(* IEC 61131-3 sources: 1326_JeddahAppartment/1326 - Jeddah Appartment - Last/PLC1, 11 files *)

(* ---- PLC1.ST ---- *)
TYPE
  TCurtainStatus : Struct
    outUP   : BOOl;
    outDW   : BOOl;
    pos     : USINT;
    normPos : USINT;
  End_Struct;
END_TYPE

TYPE
   TEnCurtain : Struct
      UP   : BOOL;
      DW   : BOOl;
      STOP : BOOL;
   End_Struct;
END_TYPE

VAR_GLOBAL CONSTANT
   numOfCurtains      : USINT := 14;
   numOfCurtains_PLC1 : USINT := 9;
   numOfCurtains_PLC2 : USINT := 5;
END_VAR

VAR_GLOBAL
  curtainsStatus  AT PLC3.DATA : Array[1..numOfCurtains] of TCurtainStatus;
  PLC1_EnCurtains AT PLC1_Curtains.DATA : Array[1..numOfCurtains_PLC1] of TEnCurtain;
  PLC2_EnCurtains AT PLC2_Curtains.DATA : Array[1..numOfCurtains_PLC2] of TEnCurtain;
END_VAR

(* ---- fbControlFCU.ST ---- *)
Type
  TFCU_Mode      : (cooling, fanOnly);
  TFCU_FanSpeed  : (auto, low, med, high);

  TFCU_Settings  : Struct
     FCU_Mode     : TFCU_Mode;
     FCU_FanSpeed : TFCU_FanSpeed;
  End_Struct
End_Type

FUNCTION_BLOCK fbControlFCU
  VAR_INPUT
  enable   : BOOL;
  mode     : TFCU_Mode;      // 0  is cooling, 1 is fan only
  fanSpeed : TFCU_FanSpeed;  // 0 auto, 1 low, 2 med, 3 high
  setTemp  : REAL;
  temp     : REAL;
  END_VAR

  VAR_OUTPUT
  FCU_Status : TFCU_Status;
  END_VAR

  VAR_IN_OUT
  valve   : BOOL;
  fanLow  : BOOL;
  fanMed  : BOOl;
  fanHigh : BOOL;
  END_VAR

  VAR
  tempDiff : REAL;
  fanRotation_tick : fbTick;
  rotationTime : Time;
  END_VAR

  tempDiff := ABS(temp - setTemp);

  if not enable then
     valve := 0;
     FCU_Status.fanSpeed := 0;
  else
     if temp >= setTemp then
        if mode = cooling then
           valve := 1;
        else
           valve := 0;
        end_if;

        if fanSpeed <> auto then
           if fanSpeed = low then
              FCU_Status.fanSpeed := 1;
           elsif fanSpeed = med then
              FCU_Status.fanSpeed := 2;
           elsif fanSpeed = high then
              FCU_Status.fanSpeed := 4;
           end_if;
        else
           if tempDiff <= 2 then
              FCU_Status.fanSpeed := 1;
           elsif tempDiff >= 2.5 and tempDiff <= 4 then
              FCU_Status.fanSpeed := 2;
           elsif tempDiff >= 4.5 then
              FCU_Status.fanSpeed := 4;
           end_if;
        end_if;

     elsif temp < setTemp - 1 then
        valve := 0;
        if mode = fanOnly and fanSpeed <> auto then
           if fanSpeed = low then
              FCU_Status.fanSpeed := 1;
           elsif fanSpeed = med then
              FCU_Status.fanSpeed := 2;
           elsif fanSpeed = high then
              FCU_Status.fanSpeed := 4;
           end_if;
        else
           FCU_Status.fanSpeed := 0;
        end_if;
     end_if;
  end_if;

  fanLow  := FCU_Status.fanSpeed.0;
  fanMed  := FCU_Status.fanSpeed.1;
  fanHigh := FCU_Status.fanSpeed.2;

  FCU_Status.onOffStatus.0 := enable;
  FCU_Status.setTemp       := REAL_TO_INT(setTemp * 100);
  FCU_Status.roomTemp      := REAL_TO_INT(temp * 100);
  FCU_Status.valve.0       := valve;

  if mode = cooling then
     FCU_Status.mode := 0;
  elsif mode = fanOnly then
     FCU_Status.mode := 1;
  end_if;

  if fanSpeed = auto then
     FCU_Status.fanSpeedCtrl := 8;
  elsif fanSpeed = low then
     FCU_Status.fanSpeedCtrl := 1;
  elsif fanSpeed = med then
     FCU_Status.fanSpeedCtrl := 2;
  elsif fanSpeed = high then
     FCU_Status.fanSpeedCtrl := 4;
  end_if;

  if FCU_Status.fanSpeed = 0 then
     FCU_Status.fanRotationVar := 0;
  elsif FCU_Status.fanSpeed = 1 then
     rotationTime := T#0.5s;
  elsif FCU_Status.fanSpeed = 2 then
     rotationTime := T#0.25s;
  elsif FCU_Status.fanSpeed = 4 then
     rotationTime := T#0.1s;
  end_if;

  fanRotation_tick(IN := FCU_Status.fanSpeed <> 0, PT := rotationTime);

  if fanRotation_tick.Q then
     FCU_Status.fanRotationVar := UINT_TO_WORD(WORD_TO_UINT(FCU_Status.fanRotationVar) + 1);
  end_if;

  if FCU_Status.fanRotationVar = 6 then
     FCU_Status.fanRotationVar := 0;
  end_if;

END_FUNCTION_BLOCK

(* ---- fbControlHotelSystem_UDP.ST ---- *)
TYPE
  THotelPacket_Head : STRUCT
    frameHeader : WORD := 16#55AA;
    frameLength : UINT;
    SystemID    : DWORD := 16#41533354;
    cmdType     : Byte := 16#0F;
    frameNo     : WORD := 16#003A;
    nBuild      : BYTE := 16#FF;
    nUnit       : BYTE := 16#FF;
    nFloor      : BYTE := 16#FF;
    nRoom       : BYTE := 16#FF;
  END_STRUCT;
  TDevTypes :  (strongRelay := 1 , weakInput := 2 , weakOutput := 3 , serviceInfo := 4, curtainNode := 5,
              RS485Switch := 6, AirCond1 := 7, AirCond2 := 8, AirCond3 := 9, RS485Card := 10, RS485Heater := 11, EX_Relay := 14,
              IR := 15, EX_LED := 16, EX_Triac := 17, EX_RGB := 18, coreCtrl := 19, WeChatLock := 20, backMusic := 21,
              roomStateDimm := 22 , PMW_OUT := 23) ;

  TCtrlType : (open := 1, close := 2);

  TDevice : STRUCT
    DevType : TDevTypes;
    DevAddress : USINT ;
    loopAddress: UINT ;
    CtrlType   : TCtrlType := open;
    CtrlContent: USINT; (*from 0 to 100*)
  END_STRUCT;

  TDevCtrl : STRUCT
    NumOfDev : USINT := 1;
    DevArr : ARRAY [1..185] OF TDevice;
  END_STRUCT;

  THotelPacket : STRUCT
    Header : THotelPacket_Head;
    Data   : TDevCtrl;
    CRC    : UINT;
  END_STRUCT;

  TServerPacket : Struct
    userCode : Array[1..4] of byte := [0,0,0,0]; // keep zeros
    heartBeat: byte := 1;    // keep 1
    IP   :  TIPadr;
    port : UINT := 61000;
  END_Struct;

  TIamServerPacket : Struct
    Header         : THotelPacket_Head := (cmdType := 1 , frameNo := 16#000E);
    serverSettings : TServerPacket;
    CRC            : UINT;
  End_Struct;

  TAllStatusPacket : struct
    Header         : THotelPacket_Head;
    CRC            : UINT;
  End_struct;
END_TYPE

TYPE
   TDeviceStatus : STRUCT
    DevType : USINT;
    DevAddress : USINT ;
    loopAddress: UINT ;
    CtrlType   : BOOL;
    CtrlContent: USINT; (*from 0 to 100*)
  END_STRUCT;
END_TYPE

Type
    TBufferIn : Array[0..1349] of usint;
END_TYPE

FUNCTION_BLOCK fbControlHotelSystem_UDP
  VAR_INPUT

  RQ : BOOL;
  sendIamServer : BOOL R_EDGE;
  getAllStatus   : BOOL R_EDGE;
  ChanCode :  UINT;
  serverSettings : TServerPacket;

  END_VAR
  VAR_IN_OUT
  packet : THotelPacket;
  CH_IN : TBufferIn;
  END_vAR

  VAR_OUTPUT

  DevicesStatus : array[1..185] of TDeviceStatus;
  SysLock , cardType , Door : BOOl;
  numOfStatusDevs : uint;
  msgSent : BOOL;
  errCode : USINT;
  errText : STRING[100];
  END_VAR
  VAR
  IamServerPacket : TIamServerPacket;
  allStatusPacket : TAllStatusPacket;
  i : uint;
  index : uint;
  startIndex : UINT := 23;
  send_UDP : fbSendTO;
  CRC {Hidden} : PTR_TO UINT;
  END_VAR
  // OLD **** max controlled devices is 185 but the channel size must be max =  1350
  // In this project the channel length is modified in order to be able to create 7 channels
  // because when we crete 7 channels with 1350 bytes then the compiler reported allocation confilct error
  if not sendIamServer and not getAllStatus then
    if packet.Data.NumOfDev <= 0 then
       errCode := 65;
       errText := 'The number of devices is zero';
    elsif packet.Data.NumOfDev > 185 then
       errCode := 66;
       errText := 'The max number of devices is exceeded';
    else
      packet.Header.frameLength := SIZEOF(packet.Header) + 3 + (usint_to_uint(packet.Data.NumOfDev) * 6);
     // Length := packet.Header.frameLength;
      if packet.Header.frameLength <> 0 then
         if packet.Data.NumOfDev < 185  then
            CRC := adr(packet.Data.DevArr[packet.data.NumOfDev+1]);
            CRC^ := CheckCRC_16(ptr := adr(packet), length := packet.Header.frameLength - 2) ;
            packet.CRC := CRC^;
         elsif packet.Data.NumOfDev = 185 then
            packet.CRC := CheckCRC_16(ptr := adr(packet), length := packet.Header.frameLength - 2);
         end_if;
      end_if;
      send_UDP(rq := RQ, chanCode := ChanCode, lenTx := packet.Header.frameLength, data := void(packet) , mesSent => msgSent , error => errCode);
      errText := GetLastComErrTxt(errCode := errCode);
    end_if;
  elsif sendIamServer then
    IamServerPacket.Header.frameLength := SIZEOF(IamServerPacket) ;
    IamServerPacket.serverSettings := serverSettings;
    IamServerPacket.CRC := CheckCRC_16(ptr := adr(IamServerPacket), length := IamServerPacket.Header.frameLength - 2);

    send_UDP(rq := true, chanCode := ChanCode, lenTx := IamServerPacket.Header.frameLength, data := void(IamServerPacket) , mesSent => msgSent , error => errCode);
    errText := GetLastComErrTxt(errCode := errCode);
  elsif getAllStatus then
    allStatusPacket.Header.cmdType := 16#0E;
    allStatusPacket.Header.frameNo := 16#0001;
    allStatusPacket.Header.frameLength := SIZEOF(allStatusPacket);
    allStatusPacket.CRC := CheckCRC_16(ptr := adr(allStatusPacket), length := allStatusPacket.Header.frameLength - 2);

    send_UDP(rq := true, chanCode := ChanCode, lenTx := allStatusPacket.Header.frameLength, data := void(allStatusPacket) , mesSent => msgSent , error => errCode);
    errText := GetLastComErrTxt(errCode := errCode);
  end_if;

  // Read Status
  startIndex := 23;

  if CH_IN[8] = 14 then
    numOfStatusDevs := usint_to_uint(CH_IN[22]);
    for i := 1 to numOfStatusDevs  do
       index := startIndex + (i-1) * 6;
       DevicesStatus[i].DevType := CH_IN[index];
       DevicesStatus[i].DevAddress := CH_IN[index+1];
       DevicesStatus[i].loopAddress := USINT_TO_UINT(CH_IN[index+2]);
       if CH_IN[index+4] = 1 then
          DevicesStatus[i].CtrlType := true;
       elsif CH_IN[index+4] = 2 then
          DevicesStatus[i].CtrlType := false;
       end_if;
       DevicesStatus[i].CtrlContent := CH_IN[index+5];
    End_For;
    SysLock := usint_to_bool(CH_IN[15]);
    cardType := usint_to_bool(CH_IN[16]);
    Door  := usint_to_bool(CH_IN[17]);

  End_if;

END_FUNCTION_BLOCK

(* ---- fbControlRoom.ST ---- *)
Type
   TOutDev : struct
     DevAddress : USINT ;
     loopAddress: UINT ;
   End_Struct
End_Type

Type
  TLightsStatus         : Array[1..17] of BOOL ;
  TOutletsStatus        : Array[1..8]  of BOOL;
  TCurtainsUpStatus     : Array[1..6]  of BOOL;
  TCurtainsDwStatus     : Array[1..6]  of BOOL;
  TCurtainsFB           : Array[1..6]  of fb_iJalousie;
  TCurtainPositWm       : Array[1..6]  OF USINT;
  TMotionSensStatus     : Array[1..4]  of BOOL;
  TSwitchStatus         : Array[1..6]  of BOOL;

  TEnLights             : Array[1..17] of BOOL ;
  TEnLightsAN           : Array[1..17] of USINT; // 1:open  2:close 0:None
  //TEnLightsAN1          : USINT;
  TEnOutlets            : Array[1..8]  of BOOL;
  TEnOutletsAN          : Array[1..8]  of USINT; // 1:open  2:close 0:None
  TEnCurtainsUp         : Array[1..6]  of BOOL;
  TEnCurtainsDW         : Array[1..6]  of BOOL;

  TlightsOutputDevs     : Array[1..17] of TOutDev;
  ToutletOutputDevs     : Array[1..8]  of TOutDev;
  TcurtainsUpOutputDevs : Array[1..6]  of TOutDev;
  TcurtainsDwOutputDevs : Array[1..6]  of TOutDev;
  TMotionSensOutputDevs : Array[1..4]  of TOutDev;
  TExRelayAdd           : ARRAY[1..2]  OF USINT;

End_Type

FUNCTION_BLOCK fbControlRoom
(*function block that send the command to RCU to control
the lights, curtains, and outlets
*)
  VAR_INPUT
    RCU_ChCode       : UINT;
   // RCU_ethAdrToSet  : TRemoteEthAdr;

   // RCU_IP_toSet     : TIPadr;

    numOfLights      : USINT;
    numOfOutlets     : USINT;
    numOfCurtains    : USINT;
    numOfMotionSens  : USINT;
    RCU_PingDone     : BOOL;

    lightsOutputDevs      : TlightsOutputDevs;
    outletOutputDevs      : ToutletOutputDevs;
    curtainsUpOutputDevs  : TcurtainsUpOutputDevs;
    curtainsDwOutputDevs  : TcurtainsDwOutputDevs;
    MotionSensOutputDevs  : TMotionSensOutputDevs;

  END_VAR
  VAR_OUTPUT
  //    CurtainPositWm   : TCurtainPositWm;

      ExRelay1_LVO : array[1..24] of TDeviceStatus;
      ExRelay2_LVO : array[1..24] of TDeviceStatus;

      SwitchUPStatus  : TSwitchStatus;
      SwitchDWStatus  : TSwitchStatus;
  END_VAR
  VAR_IN_OUT
    RCU_CH_IN     : TBufferIn;
 //   Set_IP           : BOOL;

    LightsStatus     : TLightsStatus;
    OutletsStatus    : TOutletsStatus;
  //  CurtainsUpStatus : TCurtainsUpStatus;
  //  CurtainsDwStatus : TCurtainsDwStatus;
  //  CurtainsFB       : TCurtainsFB;
    MotionSenStatus  : TMotionSensStatus;

    EnLights       : TEnLights     ;
    EnLightsAN     : TEnLightsAN   ;
   // EnLightsAN1  : TEnLightsAN1;
    EnOutlets      : TEnOutlets    ;
    EnOutletsAN    : TEnOutletsAN   ;
  //  EnCurtainsUp   : TEnCurtainsUp ;
  //  EnCurtainsDw   : TEnCurtainsDW ;

    SendIamServer : BOOL;
    GetAllStatus  : BOOL;

  END_VAR
  VAR
    RCU           : fbControlHotelSystem_UDP;
    RCU_RQ        : BOOL;
    Server_settings  : TServerPacket := (IP := [192,168,0,16])  ;
    sentPacket       : THotelPacket;
    K : USINT;
    i : UINT;
    cmd_CtrlType     : TCtrlType  ;
    cmd_CtrlContent  : USINT;
    cmd_CtrlType1    : TCtrlType  ;
    cmd_CtrlContent1 : USINT;

    TonCurtainsWait : Array[1..5]  of TON ;
    EnCurtainsWait  : Array[1..5]  of BOOL ;
    //TpCurtains      : Array[1..5]  of TPR;
    EnCurtains      : Array[1..5]  of BOOL ;
    //ReCurtainsTp    : Array[1..5]  of BOOL ;
    RTCurtains      : Array[1..5]  of R_TRIG;
    FTCurtains      : Array[1..5]  of F_TRIG;
    Up              : Array[1..5]  of BOOL ;
    Dw              : Array[1..5]  of BOOL ;
    NumOfCmd        : USINT := 1;
    RCU_Connected   : BOOL;

    RCU_Connected_RT : R_TRIG;
    RCU_Connection_TOF : TOF;
    restorStatusDone      : BOOL;
    test                  : USINT;
    PlcEthAdr             : TlocalEthAdr ;
    RCU_ChAdr             : TRemoteEthAdr;

  END_VAR

//  IF Set_IP THEN
//     SetRemoteIPaddress(rq := True , chanCode :=RCU_ChCode , ethAdr :=RCU_ethAdrToSet ) ;
//     Set_IP := 0 ;
//  END_IF;

   for i := 1 to RCU.numOfStatusDevs do

      if RCU.DevicesStatus[i].DevType = 6 and RCU.DevicesStatus[i].DevAddress = 1 then
        ExRelay1_LVO[RCU.DevicesStatus[i].loopAddress] := RCU.DevicesStatus[i];

      elsif RCU.DevicesStatus[i].DevType = 6 and RCU.DevicesStatus[i].DevAddress = 2 then
        ExRelay2_LVO[RCU.DevicesStatus[i].loopAddress] := RCU.DevicesStatus[i];
      end_if;

   End_for;

  if GetIPaddress(ethChan := ETH1 , ethAdr := PlcEthAdr) then
     Server_settings.IP := PlcEthAdr.IP ;
  end_if;

  if GetRemoteIPaddress(chanCode := RCU_ChCode, ethAdr := RCU_ChAdr) then
     Server_settings.port := RCU_ChAdr.localPort ;
  end_if;

  RCU(RQ := RCU_RQ , sendIamServer :=SendIamServer , getAllStatus := GetAllStatus , ChanCode := RCU_ChCode , serverSettings := Server_settings , packet := sentPacket, CH_IN := RCU_CH_IN);

  IF RCU.msgSent THEN
    RCU_RQ := 0 ;
    SendIamServer := 0 ;
    GetAllStatus  := 0 ;
    NumOfCmd := 1 ;
    restorStatusDone :=0;
  END_IF;

  RCU_Connection_TOF(IN := RCU_PingDone , PT :=T#1s , Q => RCU_Connected );
  RCU_Connected_RT(CLK := RCU_Connected );

  IF RCU_Connected_RT.Q THEN
    restorStatusDone :=1;
  END_IF;
  IF IS_COLD_RESTART_PLC OR IS_HOT_RESTART_PLC THEN
     GetAllStatus :=1;
  END_IF;
  IF restorStatusDone THEN
     if numOfLights > 0 then
       FOR K := 1 TO numOfLights DO
          IF LightsStatus[K] THEN
            cmd_CtrlType := open ;
            cmd_CtrlContent := 100 ;
          ELSE
            cmd_CtrlType := close ;
            cmd_CtrlContent := 0 ;
          END_IF;
          sentPacket.Data.DevArr[NumOfCmd].DevType     := EX_Relay ;
          sentPacket.Data.DevArr[NumOfCmd].DevAddress  := lightsOutputDevs[K].DevAddress;
          sentPacket.Data.DevArr[NumOfCmd].loopAddress := lightsOutputDevs[K].loopAddress ;
          sentPacket.Data.DevArr[NumOfCmd].CtrlType    := cmd_CtrlType ;
          sentPacket.Data.DevArr[NumOfCmd].CtrlContent := cmd_CtrlContent ;
          NumOfCmd := NumOfCmd + 1 ;
          test := test + 1 ;
       END_FOR;
     end_if;

     if numOfOutlets > 0 then
       FOR K := 1 TO numOfOutlets DO
          IF OutletsStatus[K] THEN
            cmd_CtrlType := open ;
            cmd_CtrlContent := 100 ;
          ELSE
            cmd_CtrlType := close ;
            cmd_CtrlContent := 0 ;
          END_IF;
          sentPacket.Data.DevArr[NumOfCmd].DevType     := EX_Relay ;
          sentPacket.Data.DevArr[NumOfCmd].DevAddress  := outletOutputDevs[K].DevAddress;
          sentPacket.Data.DevArr[NumOfCmd].loopAddress := outletOutputDevs[K].loopAddress ;
          sentPacket.Data.DevArr[NumOfCmd].CtrlType    := cmd_CtrlType ;
          sentPacket.Data.DevArr[NumOfCmd].CtrlContent := cmd_CtrlContent ;
          NumOfCmd := NumOfCmd + 1 ;
       END_FOR;
     end_if;
     sentPacket.Data.NumOfDev := NumOfCmd ;
     RCU_RQ := 1 ;
     restorStatusDone := 0;
    // GetAllStatus := 1;
  ELSE
    FOR i := 1 to RCU.numOfStatusDevs DO
       IF RCU.DevicesStatus[i].DevType = 14 THEN
         if numOfLights > 0 then
           FOR K := 1 TO numOfLights DO
             IF RCU.DevicesStatus[i].loopAddress = lightsOutputDevs[K].loopAddress AND RCU.DevicesStatus[i].DevAddress = lightsOutputDevs[K].DevAddress THEN
                lightsStatus[K] := RCU.DevicesStatus[i].CtrlType;
             END_IF;
           END_FOR;
         end_if;

         if numOfOutlets > 0 then
           FOR K := 1 TO numOfOutlets DO
             IF RCU.DevicesStatus[i].loopAddress = outletOutputDevs[K].loopAddress AND RCU.DevicesStatus[i].DevAddress = outletOutputDevs[k].DevAddress THEN
                outletsStatus[K] := RCU.DevicesStatus[i].CtrlType;
             END_IF;
           END_FOR;
         end_if;
        (* FOR K := 1 TO numOfCurtains DO
           IF RCU.DevicesStatus[i].loopAddress = curtainsUpOutputDevs[K].loopAddress AND RCU.DevicesStatus[i].DevAddress = curtainsUpOutputDevs[K].DevAddress  THEN
              CurtainsUpStatus[K] := RCU.DevicesStatus[i].CtrlType;
           END_IF;
         END_FOR;
         FOR K := 1 TO numOfCurtains DO
           IF RCU.DevicesStatus[i].loopAddress = curtainsDwOutputDevs[K].loopAddress AND RCU.DevicesStatus[i].DevAddress = curtainsDwOutputDevs[K].DevAddress THEN
              CurtainsDwStatus[K] := RCU.DevicesStatus[i].CtrlType;
           END_IF;
         END_FOR; *)

       ELSIF RCU.DevicesStatus[i].DevType = 6 THEN

         // get the status of motion sensors
         if numOfMotionSens > 0 then
           FOR K := 1 TO numOfMotionSens  DO
             IF RCU.DevicesStatus[i].loopAddress = MotionSensOutputDevs[K].loopAddress AND RCU.DevicesStatus[i].DevAddress = MotionSensOutputDevs[K].DevAddress THEN
                MotionSenStatus[K] := RCU.DevicesStatus[i].CtrlType;
             END_IF;
           END_FOR;
         end_if;

         // Get the status of switch keys from the RCU
         if numOfCurtains > 0 then
           FOR K := 1 TO numOfCurtains  DO
             IF RCU.DevicesStatus[i].loopAddress = curtainsUpOutputDevs[K].loopAddress AND RCU.DevicesStatus[i].DevAddress = curtainsUpOutputDevs[K].DevAddress THEN
                SwitchUPStatus[K] := RCU.DevicesStatus[i].CtrlType;
             END_IF;

             IF RCU.DevicesStatus[i].loopAddress = curtainsDwOutputDevs[K].loopAddress AND RCU.DevicesStatus[i].DevAddress = curtainsDwOutputDevs[K].DevAddress THEN
                SwitchDWStatus[K] := RCU.DevicesStatus[i].CtrlType;
             END_IF;
           END_FOR;
         end_if;

       END_IF;
    END_FOR;
  END_IF;

  //FOR test
  (*IF (EnLightsAN1 = 1 AND LightsStatus[1] = false) OR (EnLightsAN1 = 2 AND LightsStatus[1] = true) THEN
      EnLights[1]   := 1;
      EnLightsAN1 := 0;
  ELSE
      EnLightsAN1 :=0;
  END_IF;*)

  if numOfLights > 0 then
    FOR K := 1 TO numOfLights DO
       IF (EnLightsAN[K] = 1 AND LightsStatus[K] = false) OR (EnLightsAN[K] = 2 AND LightsStatus[K] = true) THEN
          EnLights[K]   := 1;
          EnLightsAN[K] := 0;
       ELSE
          EnLightsAN[K] :=0;
       END_IF;

       IF EnLights[K] THEN
         EnLights[K] := 0 ;
         IF lightsStatus[K] THEN
            cmd_CtrlType     := close ;
            cmd_CtrlContent  := 0 ;
         ELSE
            cmd_CtrlType     := open ;
            cmd_CtrlContent  := 100 ;
         END_IF;
         sentPacket.Data.NumOfDev := 1 ;
         sentPacket.Data.DevArr[1].DevType := EX_Relay ;
         sentPacket.Data.DevArr[1].DevAddress := lightsOutputDevs[K].DevAddress;
         sentPacket.Data.DevArr[1].loopAddress := lightsOutputDevs[K].loopAddress ;
         sentPacket.Data.DevArr[1].CtrlType := cmd_CtrlType ;
         sentPacket.Data.DevArr[1].CtrlContent := cmd_CtrlContent ;
         RCU_RQ :=1;
       END_IF;
    END_FOR;
  end_if;

  if numOfOutlets > 0 then
    FOR K := 1 TO numOfOutlets DO
       IF (EnOutletsAN[K] = 1 AND OutletsStatus[K] = false) OR (EnOutletsAN[K] = 2 AND OutletsStatus[K] = true) THEN
          EnOutlets[K]   := 1;
          EnOutletsAN[K] := 0;
       ELSE
          EnOutletsAN[K] := 0;
       END_IF;

       IF EnOutlets[K] THEN
         EnOutlets[K] := 0 ;
         IF outletsStatus[K] THEN
            cmd_CtrlType     := close ;
            cmd_CtrlContent  := 0 ;
         ELSE
            cmd_CtrlType     := open ;
            cmd_CtrlContent  := 100 ;
         END_IF;
         sentPacket.Data.NumOfDev := 1 ;
         sentPacket.Data.DevArr[1].DevType := EX_Relay ;
         sentPacket.Data.DevArr[1].DevAddress := outletOutputDevs[K].DevAddress;
         sentPacket.Data.DevArr[1].loopAddress := outletOutputDevs[K].loopAddress ;
         sentPacket.Data.DevArr[1].CtrlType := cmd_CtrlType ;
         sentPacket.Data.DevArr[1].CtrlContent := cmd_CtrlContent ;
         RCU_RQ :=1;
       END_IF;
    END_FOR;
  end_if;

   (*
   FOR K := 1 TO numOfCurtains DO
      IF ((EnCurtainsUp[K] AND Dw[K]) OR (EnCurtainsDw[K] AND Up[K])) THEN
       EnCurtains[K] := 0;
       curtainsFB[k](stop := 1  , upDwTime :=T#20s );

       sentPacket.Data.NumOfDev := 2 ;
       sentPacket.Data.DevArr[1].DevType := EX_Relay ;
       sentPacket.Data.DevArr[1].DevAddress := curtainsUpOutputDevs[K].DevAddress;
       sentPacket.Data.DevArr[1].loopAddress := curtainsUpOutputDevs[K].loopAddress ;
       sentPacket.Data.DevArr[1].CtrlType := close ;
       sentPacket.Data.DevArr[1].CtrlContent := 0 ;

       sentPacket.Data.DevArr[2].DevType := EX_Relay ;
       sentPacket.Data.DevArr[2].DevAddress := curtainsDwOutputDevs[K].DevAddress;
       sentPacket.Data.DevArr[2].loopAddress := curtainsDwOutputDevs[K].loopAddress ;
       sentPacket.Data.DevArr[2].CtrlType := close ;
       sentPacket.Data.DevArr[2].CtrlContent := 0 ;
       RCU_RQ :=1;

       Up[K] := EnCurtainsUp[K] ;
       Dw[K] := EnCurtainsDw[K] ;
       EnCurtainsUp[K] := 0;
       EnCurtainsDw[K] := 0;
       EnCurtainsWait[K] := 1;
    ELSIF (EnCurtainsUp[K] AND Dw[K] = false ) OR (EnCurtainsDw[K] AND Up[K] = false ) THEN
     //  IF curtainsFB[K].posit > 0 THEN
          Up[K] := EnCurtainsUp[K] ;
          EnCurtains[K]   := 1;
     //  ELSIF curtainsFB[K].posit < 100 THEN
          Dw[K] := EnCurtainsDw[K] ;
       //   EnCurtains[K]   := 1;
    //   END_IF;
       EnCurtainsUp[K] := 0;
       EnCurtainsDw[K] := 0;

    END_IF;

    TonCurtainsWait[K](IN := EnCurtainsWait[K] , PT := T#1s );
     IF TonCurtainsWait[K].Q THEN
       EnCurtainsWait[K] := 0;
       EnCurtains[K] := 1;
     END_IF;

     IF EnCurtains[K] THEN
        curtainsFB[K](up := CurtainsUpStatus[K] , dw := CurtainsDwStatus[K]  , upDwTime :=T#20s );
     END_IF;

     IF (curtainsFB[K].posit = 0 and curtainsFB[K].outUp) OR (curtainsFB[K].posit = 100 and curtainsFB[K].outDw) THEN
        EnCurtains[K] := 0;
        Up[K] := 0;
        Dw[K] := 0;
        curtainsFB[K](stop := 1  , upDwTime :=T#20s );
     END_IF;

     IF CurtainsFB[K].posit = 0 THEN
        CurtainPositWm[k] := 0;
     ELSIF CurtainsFB[K].posit > 0 AND CurtainsFB[K].posit < 30 THEN
        CurtainPositWm[K] := 1;
     ELSIF CurtainsFB[K].posit >= 30 AND CurtainsFB[K].posit < 60 THEN
        CurtainPositWm[K] := 2;
     ELSIF CurtainsFB[K].posit >= 60 AND CurtainsFB[K].posit < 90  THEN
        CurtainPositWm[K] := 3;
     ELSIF CurtainsFB[K].posit >= 100 THEN
        CurtainPositWm[K] := 4;
     END_IF;
     IF Up[K] THEN
        cmd_CtrlType    := open;
        cmd_CtrlContent := 100;
     ELSE
        cmd_CtrlType    := close;
        cmd_CtrlContent := 0;
     END_IF;
     IF Dw[K] THEN
        cmd_CtrlType1    := open;
        cmd_CtrlContent1 := 100;
     ELSE
        cmd_CtrlType1    := close;
        cmd_CtrlContent1 := 0;
     END_IF;
     RTCurtains[K](CLK := EnCurtains[K] ) ;
     FTCurtains[K](CLK := EnCurtains[K] ) ;
     IF RTCurtains[K].Q OR FTCurtains[K].Q THEN
       sentPacket.Data.NumOfDev := 2 ;
       sentPacket.Data.DevArr[1].DevType     := EX_Relay ;
       sentPacket.Data.DevArr[1].DevAddress  := curtainsUpOutputDevs[K].DevAddress;
       sentPacket.Data.DevArr[1].loopAddress := curtainsUpOutputDevs[K].loopAddress ;
       sentPacket.Data.DevArr[1].CtrlType    := cmd_CtrlType ;
       sentPacket.Data.DevArr[1].CtrlContent := cmd_CtrlContent ;

       sentPacket.Data.DevArr[2].DevType     := EX_Relay ;
       sentPacket.Data.DevArr[2].DevAddress  := curtainsDwOutputDevs[K].DevAddress;
       sentPacket.Data.DevArr[2].loopAddress := curtainsDwOutputDevs[K].loopAddress ;
       sentPacket.Data.DevArr[2].CtrlType    := cmd_CtrlType1 ;
       sentPacket.Data.DevArr[2].CtrlContent := cmd_CtrlContent1 ;
       RCU_RQ :=1;
     END_IF;
   END_FOR;  *)

END_FUNCTION_BLOCK

(* ---- PrgConnectHMIs.ST ---- *)
Type
  T_HMI_Info : struct
     SNo          : USINT;
     readStAdd    : UINT;
     writeStAdd   : UINT;
     readNoPoint  : UINT;
     writeNoPoint : UINT;
  End_Struct;

  //================= Read from HMI =================

  TShutterControl : struct
     Dw : WORD;
     UP : WORD;
  End_Struct;

  TFCU_Control : struct
     onOff       : WORD;
     SetTempCtrl : WORD; //  bit 0 for increment, bit 1 for decrement
     setTemp     : INT;
     fanSpeed    : WORD;
     mode        : WORD;
  End_Struct;

  T_HMI_DataRead : struct
     enLights   : Array[1..17] of WORD;
     enOutlets  : Array[1..8] of WORD;
     enShutters : Array[1..6] of TShutterControl;
     enFCUs     : Array[1..3] of TFCU_Control;
  End_Struct;

  //================= Write To HMI ==================

  TShutterStatus : struct
     Dw  : WORD;
     UP  : WORD;
     pos : WORD;
  End_Struct;

  TFCU_Status  : Struct
     onOffStatus    : WORD;
     setTemp        : INT;
     roomTemp       : INT;
     fanSpeed       : WORD;
     mode           : WORD;
     valve          : WORD;
     fanSpeedCtrl   : WORD;
     fanRotationVar : WORD;   // var for rotating the fan GIF in the HMI according to the current fan speed
  End_Struct;

  T_HMI_DataWrite : struct
     lightsStatus     : Array[1..17] of WORD;
     outletsStatus    : Array[1..8]  of WORD;
     motionSensStatus : Array[1..4]  of WORD;
     shuttersStatus   : Array[1..6]  of TShutterStatus;
     FCUs_Status      : Array[1..3]  of TFCU_Status;
  End_Struct;

End_Type

Var_Global Constant
   numOfHMIs : INT := 10;
   //HMIs_Info : Array[1..numOfHMIs] of T_HMI_Info := [()];
End_Var

Var_Global Retain
   HMIs_DataRead  : Array[1..numOfHMIs] of T_HMI_DataRead;     // Data is read from HMI
   HMIs_DataWrite : Array[1..numOfHMIs] of T_HMI_DataWrite;    // Data is written to HMI

   HMIs_Info : Array[1..numOfHMIs] of T_HMI_Info := [()];
End_Var

Var_Global
  cmdArr : Array[1..numOfHMIs * 2] of TCmdStruct;
  GrSel  : USINT ;
End_Var

PROGRAM PrgConnectHMIs
  VAR_INPUT
  END_VAR
  VAR_OUTPUT
  END_VAR
  VAR
  master : fbModbusRTUmas2;
  //cmdArr : Array[1..numOfHMIs * 2] of TCmdStruct;

  i      : INT ;
  maxCmd : USINT;

  END_VAR
  VAR_TEMP
  END_VAR

  if IS_COLD_RESTART_PLC or IS_HOT_RESTART_PLC then
     GrSel := 2;
  end_if;

  for i := 1 to numOfHMIs do
      ModbusCmd(Gr := 2, SNo := HMIs_Info[i].SNo, FNC := 3,  StAdr := HMIs_Info[i].readStAdd,   NoPoint := HMIs_Info[i].readNoPoint, PtrData := adr(HMIs_DataRead[i]), Cmd := cmdArr[i*2-1]) ;

      ModbusCmd(Gr := 2, SNo := HMIs_Info[i].SNo, FNC := 16, StAdr := HMIs_Info[i].writeStAdd , NoPoint := HMIs_Info[i].writeNoPoint, PtrData := adr(HMIs_DataWrite[i]), Cmd := cmdArr[i*2]) ;
  end_for;

  //maxCmd := INT_TO_USINT(numOfHMIs * 2);

  maxCmd := 2;
  master(EN := true, GrSel := GrSel,  MaxCmd := maxCmd , chanCode := CH2_uni , Delay := T#0.2s, Commands := cmdArr[9], MBtimeOut := T#0.5s);

END_PROGRAM

(* ---- PrgInterance.ST ---- *)
VAR_GLOBAL CONSTANT
   NumOfLightInterance      : USINT := 6;
   NumOfOutletInterance     : USINT := 2;
   NumOfCurtainInterance    : USINT := 0;
   NumOfMotionSensInterance : USINT := 1;
   NumOfFCUsInterance       : USINT := 0;
   NumOfHMIsInterance       : USINT := 1;
END_VAR

VAR_GLOBAL RETAIN
   lightsStatusInterance  {PUBLIC_API} : TLightsStatus;
   outletsStatusInterance {PUBLIC_API} : TOutletsStatus;
 (*  setTempFCU_Interance  : Array[1..NumOfFCUsInterance] of REAL := [20];
  *)

END_VAR

PROGRAM PrgInterance

  VAR
  //WebMaker
  lightsSelect   : BOOL;
  socketsSelect  : BOOL;
  shuttersSelect : BOOL;
  AC_Select      : BOOL;
  navSelect      : usint;

  //RCU
  RCU_ethAdr   : TRemoteEthAdr;
  RCU_IP : TIPadr := [192, 168, 0, 23];
  RCU_Ch_localPort : UINT;
  Set_IP           : BOOL;
  GetAllStatus  : BOOL;
  SendIamServer : BOOL;

  //controlRoom
  controlRoom   : fbControlRoom ;
  lightsOutputDevs     : TlightsOutputDevs     := [(DevAddress := 1 , loopAddress := 1),(DevAddress := 1 , loopAddress := 2),
                                                   (DevAddress := 1 , loopAddress := 3),(DevAddress := 1 , loopAddress := 4),
                                                   (DevAddress := 1 , loopAddress := 5),(DevAddress := 1 , loopAddress := 6)];

  outletOutputDevs     : ToutletOutputDevs     := [(DevAddress := 1 , loopAddress := 7)];

  (*curtainsUpOutputDevs : TcurtainsUpOutputDevs := [(DevAddress := 1 , loopAddress := 8)];
  curtainsDwOutputDevs : TcurtainsDwOutputDevs := [(DevAddress := 1 , loopAddress := 9)];*)

  motionSensOutputDevs : TMotionSensOutputDevs := [(DevAddress := 1 , loopAddress := 1)];

  EnLights                            : TEnLights     ;
  EnLightsAN       {PUBLIC_API}       : TEnLightsAN   ;
  EnOutlets                           : TEnOutlets    ;
  EnOutletsAN      {PUBLIC_API}       : TEnOutletsAN  ;
  EnCurtainsUp     {PUBLIC_API}       : TEnCurtainsUp ;
  EnCurtainsDw     {PUBLIC_API}       : TEnCurtainsDW ;
   //EnLightsInteranceAN1  {PUBLIC_API}      : TEnLightsAN1    ;
   //stLightsInteranceAN  {PUBLIC_API}       : BOOL     ;
  //curtainsFB       : TCurtainsFB;
  //CurtainPositWm   : TCurtainPositWm;

  //
  enLights_RT  : Array[1..NumOfHMIsInterance,1..NumOfLightInterance] of R_TRIG;
  enLights_FT  : Array[1..NumOfHMIsInterance,1..NumOfLightInterance] of F_TRIG;

  enOutlets_RT : Array[1..NumOfHMIsInterance,1..NumOfOutletInterance] of R_TRIG;
  enOutlets_FT : Array[1..NumOfHMIsInterance,1..NumOfOutletInterance] of F_TRIG;
  (*
  enCurtainsUP_RT : Array[1..NumOfHMIsInterance,1..NumOfCurtainInterance] of R_TRIG;
  enCurtainsUP_FT : Array[1..NumOfHMIsInterance,1..NumOfCurtainInterance] of F_TRIG;

  enCurtainsDW_RT : Array[1..NumOfHMIsInterance,1..NumOfCurtainInterance] of R_TRIG;
  enCurtainsDW_FT : Array[1..NumOfHMIsInterance,1..NumOfCurtainInterance] of F_TRIG; *)

  //
  i , j : USINT;
  afterRestart_TP : TP;
  afterRestart_TP_FT : F_TRIG;

  //
  motionSensStatus                : TMotionSensStatus;
  CurtainsUpStatus   {PUBLIC_API} : TCurtainsUpStatus;
  CurtainsDwStatus   {PUBLIC_API} : TCurtainsDwStatus;

  // FCU VARS
  (*FCU          : Array[1..NumOfFCUsInterance] of fbControlFCU;
  enableFCU    : Array[1..NumOfFCUsInterance] of BOOL;
  settingsFCU  : Array[1..NumOfFCUsInterance] of TFCU_Settings;

  //modeFCU      : Array[1..NumOfFCUsInterance] of TFCU_Mode;
  //fanSpeedFCU  : Array[1..NumOfFCUsInterance] of TFCU_FanSpeed;

  enFCUs_FT    : Array[1..NumOfHMIsInterance,1..NumOfFCUsInterance] of F_TRIG;
  enFCUs_RT    : Array[1..NumOfHMIsInterance,1..NumOfFCUsInterance] of R_TRIG;

  enFanHigh_RT : Array[1..NumOfHMIsInterance,1..NumOfFCUsInterance] of R_TRIG;
  enFanMed_RT  : Array[1..NumOfHMIsInterance,1..NumOfFCUsInterance] of R_TRIG;
  enFanLow_RT  : Array[1..NumOfHMIsInterance,1..NumOfFCUsInterance] of R_TRIG;
  enFanAuto_RT : Array[1..NumOfHMIsInterance,1..NumOfFCUsInterance] of R_TRIG;

  enFCUCool_RT    : Array[1..NumOfHMIsInterance,1..NumOfFCUsInterance] of R_TRIG;
  enFCUFanOnly_RT : Array[1..NumOfHMIsInterance,1..NumOfFCUsInterance] of R_TRIG;

  enSetTempIncr_RT : Array[1..NumOfHMIsInterance,1..NumOfFCUsInterance] of R_TRIG;
  enSetTempIncr_FT : Array[1..NumOfHMIsInterance,1..NumOfFCUsInterance] of F_TRIG;

  enSetTempDecr_RT : Array[1..NumOfHMIsInterance,1..NumOfFCUsInterance] of R_TRIG;
  enSetTempDecr_FT : Array[1..NumOfHMIsInterance,1..NumOfFCUsInterance] of F_TRIG;  *)

  //HMIs[1..num
  HMI_Index : USINT;
  RCU_Index : USINT;
  HMI_Addresses : Array[1..NumOfHMIsInterance] of USINT := [1];

  END_VAR

  if navSelect = 0 then
     lightsSelect   := 1;
     socketsSelect  := 0;

  elsif navSelect = 1 then
     lightsSelect   := 0;
     socketsSelect  := 1;
  end_if;

  HMI_Index := 1;
  RCU_Index := 1;

  if GetRemoteIPaddress(chanCode := Eth1_uni0, ethAdr := RCU_ethAdr) then
     RCUs_IPs[RCU_Index] := RCU_ethAdr.remoteIP;
  end_if;

  HMIs_Info[HMI_Index].SNo := HMI_Addresses[1];
  HMIs_Info[HMI_Index].readStAdd  := 131;
  HMIs_Info[HMI_Index].writeStAdd := 191;
  HMIs_Info[HMI_Index].readNoPoint  := SIZEOF(HMIs_DataRead[HMI_Index]) / 2;
  HMIs_Info[HMI_Index].writeNoPoint := SIZEOF(HMIs_DataWrite[HMI_Index]) / 2;

  for i := 1 to NumOfHMIsInterance-1 do
    HMIs_Info[HMI_Index+i] := HMIs_Info[HMI_Index];
    HMIs_Info[HMI_Index+i].SNo := HMI_Addresses[i+1];
  end_for;

  afterRestart_TP(IN := IS_COLD_RESTART_PLC or IS_HOT_RESTART_PLC, PT := T#2s );
  afterRestart_TP_FT(CLK := afterRestart_TP.Q);

  if afterRestart_TP_FT.Q then
     SendIamServer := 1;
  end_if;

  controlRoom(RCU_ChCode := ETH1_uni0 , RCU_PingDone := RCUs_PingDone[RCU_Index],
              numOfLights := NumOfLightInterance , numOfOutlets := NumOfOutletInterance , numOfCurtains := 0, numOfMotionSens := NumOfMotionSensInterance,
              lightsOutputDevs := lightsOutputDevs , outletOutputDevs := outletOutputDevs ,
              RCU_CH_IN := void(ETH1_uni0_IN) , LightsStatus := lightsStatusInterance ,OutletsStatus := outletsStatusInterance, MotionSenStatus := motionSensStatus,
              EnLights := EnLights , EnLightsAN := EnLightsAN , EnOutlets := EnOutlets ,EnOutletsAN :=EnOutletsAN ,
              SendIamServer := SendIamServer , GetAllStatus := GetAllStatus);

              //stLightsInteranceAN := lightsStatusInterance[1];

   for i := 1 to NumOfLightInterance do
       HMIs_DataWrite[HMI_Index].lightsStatus[i] := BOOL_TO_WORD(lightsStatusInterance[i]);
   end_for;

   for i := 1 to NumOfOutletInterance do
       HMIs_DataWrite[HMI_Index].outletsStatus[i] := BOOL_TO_WORD(outletsStatusInterance[i]);
   end_for;

   for i := 1 to NumOfMotionSensInterance do
       HMIs_DataWrite[HMI_Index].motionSensStatus[i] := BOOL_TO_WORD(motionSensStatus[i]);
   end_for;

   for j := 1 to NumOfHMIsInterance do
     for i := 1 to NumOfLightInterance do

         enLights_RT[j,i](CLK := HMIs_DataRead[HMI_Index + j - 1].enLights[i]);

         enLights_FT[j,i](CLK := HMIs_DataRead[HMI_Index + j - 1].enLights[i]);

         if enLights_RT[j,i].Q or enLights_FT[j,i].Q then
            EnLights[i] := 1;
         end_if;
     end_for;
   end_for;

   for j := 1 to NumOfHMIsInterance do
     for i := 1 to NumOfOutletInterance do

         enOutlets_RT[j,i](CLK := HMIs_DataRead[HMI_Index + j - 1].enOutlets[i]);

         enOutlets_FT[j,i](CLK := HMIs_DataRead[HMI_Index + j - 1].enOutlets[i]);

         if enOutlets_RT[j,i].Q or enOutlets_FT[j,i].Q then
            EnOutlets[i] := 1;
         end_if;
     end_for;
   end_for;

END_PROGRAM

(* ---- prgMain.ST ---- *)
Var_Global Constant
   numOfRCUS : INT := 5;
End_Var

Var_Global Retain
   RCUs_IPs : Array[1..numOfRCUS] of TIPAdr := [[192,168,0,23],
                                                [192,168,0,15],
                                                [192,168,0,17],
                                                [192,168,0,109],
                                                [192,168,0,110]];
End_Var

Var_Global
   RCUs_PingDone : array[1..numOfRCUS] of BOOL;
End_Var

PROGRAM prgMain
  VAR_INPUT
  END_VAR
  VAR_OUTPUT
  END_VAR
  VAR
  // Check RCUs connection
  ping     : fbPingIP ;
  pingInfo : T_PING_INFO;
  tick     : fbTick;
  pingSwitch : INT;
  IP        : TIPadr;

  //

  END_VAR

  // check the connection of all RCUs

  tick(IN := 1, PT :=T#1.2s );
  if tick.Q then
     pingSwitch :=  pingSwitch + 1;
  end_if;

  if pingSwitch = numOfRCUS then
     pingSwitch := 0;
  end_if;

  if pingSwitch >= 0 and pingSwitch < numOfRCUS then
     IP := RCUs_IPs[pingSwitch + 1];
  end_if;

  ping(rqPing := tick.Q , hostIP := IP , ttl := 255 , timeLimit :=T#1s ,  pingInfo := pingInfo );

  if pingSwitch >= 0 and pingSwitch < numOfRCUS then
    IF ping.done THEN
       RCUs_PingDone[pingSwitch + 1] :=1;
    END_IF;
    IF ping.busy or ping.err THEN
       RCUs_PingDone[pingSwitch + 1] :=0;
    END_IF;
  end_if;

END_PROGRAM

(* ---- PrgMajles.ST ---- *)
VAR_GLOBAL CONSTANT
   NumOfLightMajles      : USINT := 15;
   NumOfOutletMajles     : USINT := 1;
   NumOfCurtainMajles    : USINT := 5;
   NumOfMotionSensMajles : USINT := 1;
   NumOfFCUsMajles       : USINT := 2;
   NumOfHMIsMajles       : USINT := 4;
END_VAR

VAR_GLOBAL RETAIN
   lightsStatusMajles  {PUBLIC_API} : TLightsStatus;
   outletsStatusMajles {PUBLIC_API} : TOutletsStatus;
   setTempFCU_Majles  : Array[1..NumOfFCUsMajles] of REAL := [20, 20];

END_VAR

PROGRAM PrgMajles

  VAR
  //WebMaker
  lightsSelect   : BOOL;
  socketsSelect  : BOOL;
  shuttersSelect : BOOL;
  AC_Select      : BOOL;
  navSelect      : usint;

  //RCU
  RCU1_ethAdr   : TRemoteEthAdr;
  RCU2_ethAdr   : TRemoteEthAdr;

  RCU_IP : TIPadr := [192, 168, 0, 23];
  RCU_Ch_localPort : UINT;
  Set_IP           : BOOL;
  GetAllStatus  : BOOL;
  SendIamServer : BOOL;

  //controlRoom
  controlRoomRCU1   : fbControlRoom ;
  controlRoomRCU2   : fbControlRoom ;

  lightsOutputDevs     : TlightsOutputDevs     := [(DevAddress := 1 , loopAddress := 1),(DevAddress := 1 , loopAddress := 2),(DevAddress := 1 , loopAddress := 3),
                                                   (DevAddress := 1 , loopAddress := 4),(DevAddress := 1 , loopAddress := 5),(DevAddress := 1 , loopAddress := 6),
                                                   (DevAddress := 1 , loopAddress := 7),(DevAddress := 1 , loopAddress := 8),(DevAddress := 1 , loopAddress := 9),
                                                   (DevAddress := 1 , loopAddress := 10),(DevAddress := 2 , loopAddress := 1),(DevAddress := 2 , loopAddress := 2),
                                                   (DevAddress := 2 , loopAddress := 3),(DevAddress := 2 , loopAddress := 4),(DevAddress := 2 , loopAddress := 5)];

  outletOutputDevsRCU1 : ToutletOutputDevs     := [(DevAddress := 2 , loopAddress := 6)];

  outletOutputDevsRCU2 : ToutletOutputDevs ;

  curtainsUpOutputDevs : TcurtainsUpOutputDevs := [(DevAddress := 1 , loopAddress := 2),(DevAddress := 1 , loopAddress := 4),(DevAddress := 1 , loopAddress := 6),
                                                   (DevAddress := 1 , loopAddress := 8),(DevAddress := 2 , loopAddress := 1)];

  curtainsDwOutputDevs : TcurtainsDwOutputDevs := [(DevAddress := 1 , loopAddress := 3),(DevAddress := 1 , loopAddress := 5),(DevAddress := 1 , loopAddress := 7),
                                                   (DevAddress := 1 , loopAddress := 9),(DevAddress := 2 , loopAddress := 2)];

  motionSensOutputDevs : TMotionSensOutputDevs := [(DevAddress := 1 , loopAddress := 1)];

  EnLights                            : TEnLights     ;
  EnLightsAN       {PUBLIC_API}       : TEnLightsAN   ;
  EnOutlets                           : TEnOutlets    ;
  EnOutletsAN      {PUBLIC_API}       : TEnOutletsAN  ;
  EnCurtainsUp     {PUBLIC_API}       : TEnCurtainsUp ;
  EnCurtainsDw     {PUBLIC_API}       : TEnCurtainsDW ;

  //
  enLights_RT  : Array[1..NumOfHMIsMajles,1..NumOfLightMajles] of R_TRIG;
  enLights_FT  : Array[1..NumOfHMIsMajles,1..NumOfLightMajles] of F_TRIG;

  enOutlets_RT : Array[1..NumOfHMIsMajles,1..NumOfOutletMajles] of R_TRIG;
  enOutlets_FT : Array[1..NumOfHMIsMajles,1..NumOfOutletMajles] of F_TRIG;

  // HMIs
  enCurtainsUP_RT : Array[1..NumOfHMIsMajles,1..NumOfCurtainMajles] of R_TRIG;
  enCurtainsUP_FT : Array[1..NumOfHMIsMajles,1..NumOfCurtainMajles] of F_TRIG;

  enCurtainsDW_RT : Array[1..NumOfHMIsMajles,1..NumOfCurtainMajles] of R_TRIG;
  enCurtainsDW_FT : Array[1..NumOfHMIsMajles,1..NumOfCurtainMajles] of F_TRIG;

  // RCU Switches
  enCurtainsUP_SW_RT : Array[1..NumOfCurtainMajles] of R_TRIG;
  enCurtainsUP_SW_FT : Array[1..NumOfCurtainMajles] of F_TRIG;

  enCurtainsDW_SW_RT : Array[1..NumOfCurtainMajles] of R_TRIG;
  enCurtainsDW_SW_FT : Array[1..NumOfCurtainMajles] of F_TRIG;

  // GUI
  enCurtainsUP_GUI : Array[1..NumOfCurtainMajles] of BOOL;
  enCurtainsDW_GUI : Array[1..NumOfCurtainMajles] of BOOL;

  CurtStatus_Index : USINT;
  CurtEn_Index     : USINT;

  //
  i , j : USINT;
  afterRestart_TP : TP;
  afterRestart_TP_FT : F_TRIG;

  //
  motionSensStatus                : TMotionSensStatus;
  CurtainsUpStatus   {PUBLIC_API} : TCurtainsUpStatus;
  CurtainsDwStatus   {PUBLIC_API} : TCurtainsDwStatus;

  // FCU VARS
  FCU          : Array[1..NumOfFCUsMajles] of fbControlFCU;
  enableFCU    : Array[1..NumOfFCUsMajles] of BOOL;
  settingsFCU  : Array[1..NumOfFCUsMajles] of TFCU_Settings;

  //modeFCU      : Array[1..NumOfFCUsMajles] of TFCU_Mode;
  //fanSpeedFCU  : Array[1..NumOfFCUsMajles] of TFCU_FanSpeed;

  enFCUs_FT    : Array[1..NumOfHMIsMajles,1..NumOfFCUsMajles] of F_TRIG;
  enFCUs_RT    : Array[1..NumOfHMIsMajles,1..NumOfFCUsMajles] of R_TRIG;

  enFanHigh_RT : Array[1..NumOfHMIsMajles,1..NumOfFCUsMajles] of R_TRIG;
  enFanMed_RT  : Array[1..NumOfHMIsMajles,1..NumOfFCUsMajles] of R_TRIG;
  enFanLow_RT  : Array[1..NumOfHMIsMajles,1..NumOfFCUsMajles] of R_TRIG;
  enFanAuto_RT : Array[1..NumOfHMIsMajles,1..NumOfFCUsMajles] of R_TRIG;

  enFCUCool_RT    : Array[1..NumOfHMIsMajles,1..NumOfFCUsMajles] of R_TRIG;
  enFCUFanOnly_RT : Array[1..NumOfHMIsMajles,1..NumOfFCUsMajles] of R_TRIG;

  enSetTempIncr_RT : Array[1..NumOfHMIsMajles,1..NumOfFCUsMajles] of R_TRIG;
  enSetTempIncr_FT : Array[1..NumOfHMIsMajles,1..NumOfFCUsMajles] of F_TRIG;

  enSetTempDecr_RT : Array[1..NumOfHMIsMajles,1..NumOfFCUsMajles] of R_TRIG;
  enSetTempDecr_FT : Array[1..NumOfHMIsMajles,1..NumOfFCUsMajles] of F_TRIG;

  //HMIs[1..num
  HMI_Index : USINT;
  RCU_Index : USINT;
  HMI_Addresses : Array[1..NumOfHMIsMajles] of USINT := [12, 13, 14, 15];

  END_VAR

   if navSelect = 0 then
     lightsSelect   := 1;
     socketsSelect  := 0;
     shuttersSelect := 0;
     AC_Select      := 0;
  elsif navSelect = 1 then
     lightsSelect   := 0;
     socketsSelect  := 1;
     shuttersSelect := 0;
     AC_Select      := 0;
  elsif navSelect = 2 then
     lightsSelect   := 0;
     socketsSelect  := 0;
     shuttersSelect := 1;
     AC_Select      := 0;
  elsif navSelect = 3 then
     lightsSelect   := 0;
     socketsSelect  := 0;
     shuttersSelect := 0;
     AC_Select      := 1;
  end_if;

   HMI_Index := 1;
   RCU_Index := 1;
   CurtStatus_Index := 1;
   CurtEn_Index  := 1;

   if GetRemoteIPaddress(chanCode := Eth1_uni0, ethAdr := RCU1_ethAdr) then
     RCUs_IPs[RCU_Index] := RCU1_ethAdr.remoteIP;
   end_if;

   if GetRemoteIPaddress(chanCode := Eth1_uni1, ethAdr := RCU2_ethAdr) then
     RCUs_IPs[RCU_Index + 1] := RCU2_ethAdr.remoteIP;
   end_if;

  HMIs_Info[HMI_Index].SNo := HMI_Addresses[1];
  HMIs_Info[HMI_Index].readStAdd  := 1;
  HMIs_Info[HMI_Index].writeStAdd := 61;
  HMIs_Info[HMI_Index].readNoPoint  := SIZEOF(HMIs_DataRead[HMI_Index]) / 2;
  HMIs_Info[HMI_Index].writeNoPoint := SIZEOF(HMIs_DataWrite[HMI_Index]) / 2;

  for i := 1 to NumOfHMIsMajles-1 do
    HMIs_Info[HMI_Index+i] := HMIs_Info[HMI_Index];
    HMIs_Info[HMI_Index+i].SNo := HMI_Addresses[i+1];
  end_for;

  afterRestart_TP(IN := IS_COLD_RESTART_PLC or IS_HOT_RESTART_PLC, PT := T#2s );
  afterRestart_TP_FT(CLK := afterRestart_TP.Q);

  if afterRestart_TP_FT.Q then
     SendIamServer := 1;
  end_if;

  controlRoomRCU1(RCU_ChCode := ETH1_uni0 , RCU_PingDone := RCUs_PingDone[RCU_Index],
              numOfLights := NumOfLightMajles , numOfOutlets := NumOfOutletMajles , numOfCurtains := 0, numOfMotionSens := NumOfMotionSensMajles,
              lightsOutputDevs := lightsOutputDevs , outletOutputDevs := outletOutputDevsRCU1 ,
              curtainsUpOutputDevs := curtainsUpOutputDevs , curtainsDwOutputDevs := curtainsDwOutputDevs,
              RCU_CH_IN := void(ETH1_uni0_IN) , LightsStatus := lightsStatusMajles ,OutletsStatus := outletsStatusMajles, MotionSenStatus := motionSensStatus,
              EnLights := EnLights , EnLightsAN := EnLightsAN , EnOutlets := EnOutlets ,EnOutletsAN :=EnOutletsAN ,
              SendIamServer := SendIamServer , GetAllStatus := GetAllStatus );

  controlRoomRCU2(RCU_ChCode := ETH1_uni1 , RCU_PingDone := RCUs_PingDone[RCU_Index + 1],
              numOfLights := 0 , numOfOutlets := 0 , numOfCurtains := NumOfCurtainMajles, numOfMotionSens := 0,
              outletOutputDevs := outletOutputDevsRCU2,
              curtainsUpOutputDevs := curtainsUpOutputDevs , curtainsDwOutputDevs := curtainsDwOutputDevs,
              RCU_CH_IN := void(ETH1_uni1_IN) , LightsStatus := lightsStatusMajles ,OutletsStatus := void(outletsStatusMajles[6]), MotionSenStatus := motionSensStatus,
              EnLights := EnLights , EnLightsAN := EnLightsAN , EnOutlets := void(EnOutlets[6]) ,EnOutletsAN := void(EnOutletsAN[6]) ,
              SendIamServer := SendIamServer , GetAllStatus := GetAllStatus );

              //stLightsMajlesAN := lightsStatusMajles[1];

   FCU[1](enable := enableFCU[1], mode := settingsFCU[1].FCU_Mode, fanSpeed := settingsFCU[1].FCU_FanSpeed, setTemp := setTempFCU_Majles[1], temp := FCU_Temp_Majles1, valve := FCU_valve_Majles1, fanLow := FCU_fanLow_Majles1,
                 fanMed := FCU_fanMed_Majles1, fanHigh := FCU_fanHigh_Majles1);

   FCU[2](enable := enableFCU[1], mode := settingsFCU[1].FCU_Mode, fanSpeed := settingsFCU[1].FCU_FanSpeed, setTemp := setTempFCU_Majles[1], temp := FCU_Temp_Majles1, valve := FCU_valve_Majles2, fanLow := FCU_fanLow_Majles2,
                 fanMed := FCU_fanMed_Majles2, fanHigh := FCU_fanHigh_Majles2);

   for i := 1 to NumOfLightMajles do
       HMIs_DataWrite[HMI_Index].lightsStatus[i] := BOOL_TO_WORD(lightsStatusMajles[i]);
   end_for;

   for i := 1 to NumOfOutletMajles do
       HMIs_DataWrite[HMI_Index].outletsStatus[i] := BOOL_TO_WORD(outletsStatusMajles[i]);
   end_for;

   for i := 1 to NumOfMotionSensMajles do
       HMIs_DataWrite[HMI_Index].motionSensStatus[i] := BOOL_TO_WORD(motionSensStatus[i]);
   end_for;

   for i := 1 to NumOfFCUsMajles do
      HMIs_DataWrite[HMI_Index].FCUs_Status[i] := FCU[i].FCU_Status;
   end_for;

   if NumOfCurtainMajles > 0 then
      for i := 1 to NumOfCurtainMajles do
          HMIs_DataWrite[HMI_Index].shuttersStatus[i].UP.0 := curtainsStatus[CurtStatus_Index - 1 + i].outUP;
          HMIs_DataWrite[HMI_Index].shuttersStatus[i].Dw.0 := curtainsStatus[CurtStatus_Index - 1 + i].outDW;
          HMIs_DataWrite[HMI_Index].shuttersStatus[i].pos  := USINT_TO_WORD(curtainsStatus[CurtStatus_Index - 1 + i].normPos);
      end_for;
   end_if;

   for i := 1 to NumOfHMIsMajles-1 do
     HMIs_DataWrite[HMI_Index+i] := HMIs_DataWrite[HMI_Index];
   end_for;

   for j := 1 to NumOfHMIsMajles do
     for i := 1 to NumOfLightMajles do

         enLights_RT[j,i](CLK := HMIs_DataRead[HMI_Index + j - 1].enLights[i]);

         enLights_FT[j,i](CLK := HMIs_DataRead[HMI_Index + j - 1].enLights[i]);

         if enLights_RT[j,i].Q or enLights_FT[j,i].Q then
            EnLights[i] := 1;
         end_if;
     end_for;
   end_for;

   for j := 1 to NumOfHMIsMajles do
     for i := 1 to NumOfOutletMajles do

         enOutlets_RT[j,i](CLK := HMIs_DataRead[HMI_Index + j - 1].enOutlets[i]);

         enOutlets_FT[j,i](CLK := HMIs_DataRead[HMI_Index + j - 1].enOutlets[i]);

         if enOutlets_RT[j,i].Q or enOutlets_FT[j,i].Q then
            EnOutlets[i] := 1;
         end_if;
     end_for;
   end_for;

   for j := 1 to NumOfHMIsMajles do
     for i := 1 to NumOfCurtainMajles do

         enCurtainsUP_RT[j,i](CLK := HMIs_DataRead[HMI_Index + j - 1].enShutters[i].UP.0);

         enCurtainsUP_FT[j,i](CLK := HMIs_DataRead[HMI_Index + j - 1].enShutters[i].UP.0);

         enCurtainsDW_RT[j,i](CLK := HMIs_DataRead[HMI_Index + j - 1].enShutters[i].Dw.0);

         enCurtainsDW_FT[j,i](CLK := HMIs_DataRead[HMI_Index + j - 1].enShutters[i].Dw.0);

         //
         enCurtainsUP_SW_RT[i](CLK := controlRoomRCU2.SwitchUPStatus[i]);
         enCurtainsUP_SW_FT[i](CLK := controlRoomRCU2.SwitchUPStatus[i]);

         enCurtainsDW_SW_RT[i](CLK := controlRoomRCU2.SwitchDWStatus[i]);
         enCurtainsDW_SW_FT[i](CLK := controlRoomRCU2.SwitchDWStatus[i]);

         if  enCurtainsUP_RT[j,i].Q  or enCurtainsUP_FT[j,i].Q or enCurtainsUP_SW_RT[i].Q or enCurtainsUP_SW_FT[i].Q then
             enCurtainsUP_GUI[i] := 1;
         end_if;

         if  enCurtainsDW_RT[j,i].Q  or enCurtainsDW_FT[j,i].Q or enCurtainsDW_SW_RT[i].Q or enCurtainsDW_SW_FT[i].Q then
             enCurtainsDW_GUI[i] := 1;
         end_if;

         // if up button is pressed and the curtain is not moving up

         if enCurtainsUP_GUI[i] and not curtainsStatus[CurtStatus_Index - 1 + i].outUP then
             PLC1_EnCurtains[CurtEn_Index - 1 + i].UP   := 1;
             PLC1_EnCurtains[CurtEn_Index - 1 + i].DW   := 0;
             PLC1_EnCurtains[CurtEn_Index - 1 + i].STOP := 0;

             enCurtainsUP_GUI[i] := 0;
         end_if;

         // if up button is pressed and the curtain is moving up

         if enCurtainsUP_GUI[i] and curtainsStatus[CurtStatus_Index - 1 + i].outUP then
             PLC1_EnCurtains[CurtEn_Index - 1 + i].UP   := 0;
             PLC1_EnCurtains[CurtEn_Index - 1 + i].DW   := 0;
             PLC1_EnCurtains[CurtEn_Index - 1 + i].STOP := 1;

             enCurtainsUP_GUI[i] := 0;
         end_if;

          // if down button is pressed and the curtain is not moving down

         if enCurtainsDW_GUI[i] and not curtainsStatus[CurtStatus_Index - 1 + i].outDW then
             PLC1_EnCurtains[CurtEn_Index - 1 + i].UP   := 0;
             PLC1_EnCurtains[CurtEn_Index - 1 + i].DW   := 1;
             PLC1_EnCurtains[CurtEn_Index - 1 + i].STOP := 0;

             enCurtainsDW_GUI[i] := 0;
         end_if;

         // if down button is pressed and the curtain is moving down

         if enCurtainsDW_GUI[i] and curtainsStatus[CurtStatus_Index - 1 + i].outDW then
             PLC1_EnCurtains[CurtEn_Index - 1 + i].UP   := 0;
             PLC1_EnCurtains[CurtEn_Index - 1 + i].DW   := 0;
             PLC1_EnCurtains[CurtEn_Index - 1 + i].STOP := 1;

             enCurtainsDW_GUI[i] := 0;
         end_if;

     end_for;
   end_for;

   for j := 1 to NumOfHMIsMajles do
      for i := 1 to NumOfFCUsMajles do
          enFCUs_FT[j,i](CLK := HMIs_DataRead[HMI_Index + j - 1].enFCUs[i].onOff);
          enFCUs_RT[j,i](CLK := HMIs_DataRead[HMI_Index + j - 1].enFCUs[i].onOff);

          if enFCUs_FT[j,i].Q then
             enableFCU[i] := 0;
          end_if;
          if enFCUs_RT[j,i].Q then
             enableFCU[i] := 1;
          end_if;

          enFanAuto_RT[j,i](CLK := (HMIs_DataRead[HMI_Index + j - 1].enFCUs[i].fanSpeed = 8));
          enFanLow_RT[j,i](CLK := HMIs_DataRead[HMI_Index + j - 1].enFCUs[i].fanSpeed.0);
          enFanMed_RT[j,i](CLK := HMIs_DataRead[HMI_Index + j - 1].enFCUs[i].fanSpeed.1);
          enFanHigh_RT[j,i](CLK := HMIs_DataRead[HMI_Index + j - 1].enFCUs[i].fanSpeed.2);

          if enFanAuto_RT[j,i].Q then
             settingsFCU[i].FCU_FanSpeed := auto;
          end_if;
          if enFanLow_RT[j,i].Q then
             settingsFCU[i].FCU_FanSpeed := low;
          end_if;
          if enFanMed_RT[j,i].Q then
             settingsFCU[i].FCU_FanSpeed := med;
          end_if;
          if enFanHigh_RT[j,i].Q then
             settingsFCU[i].FCU_FanSpeed := high;
          end_if;

          enFCUCool_RT[j,i](CLK := (HMIs_DataRead[HMI_Index + j - 1].enFCUs[i].mode = 0));
          enFCUFanOnly_RT[j,i](CLK := HMIs_DataRead[HMI_Index + j - 1].enFCUs[i].mode.0);

          if enFCUCool_RT[j,i].Q then
             settingsFCU[i].FCU_Mode := cooling;
          end_if;
          if enFCUFanOnly_RT[j,i].Q then
             settingsFCU[i].FCU_Mode := fanOnly;
          end_if;

          enSetTempIncr_RT[j,i](CLK := HMIs_DataRead[HMI_Index + j - 1].enFCUs[i].SetTempCtrl.0);
          enSetTempIncr_FT[j,i](CLK := HMIs_DataRead[HMI_Index + j - 1].enFCUs[i].SetTempCtrl.0);

          if enSetTempIncr_RT[j,i].Q or enSetTempIncr_FT[j,i].Q then
             setTempFCU_Majles[j] := setTempFCU_Majles[j] + 0.5;
          end_if;

          enSetTempDecr_RT[j,i](CLK := HMIs_DataRead[HMI_Index + j - 1].enFCUs[i].SetTempCtrl.1);
          enSetTempDecr_FT[j,i](CLK := HMIs_DataRead[HMI_Index + j - 1].enFCUs[i].SetTempCtrl.1);

          if enSetTempDecr_RT[j,i].Q or enSetTempDecr_FT[j,i].Q then
             setTempFCU_Majles[j] := setTempFCU_Majles[j] - 0.5;
          end_if;

      end_for;
   end_for;

END_PROGRAM

(* ---- PrgRoom1.ST ---- *)
VAR_GLOBAL CONSTANT
   NumOfLightRoom1      : USINT := 5;
   NumOfOutletRoom1     : USINT := 1;
   NumOfCurtainRoom1    : USINT := 1;
   NumOfMotionSensRoom1 : USINT := 2;
   NumOfFCUsRoom1       : USINT := 1;
   NumOfHMIsRoom1       : USINT := 2;
END_VAR

VAR_GLOBAL RETAIN
   lightsStatusRoom1  {PUBLIC_API} : TLightsStatus;
   outletsStatusRoom1 {PUBLIC_API} : TOutletsStatus;
   setTempFCU_Room1  : Array[1..NumOfFCUsRoom1] of REAL := [20];
END_VAR

PROGRAM PrgRoom1

  VAR
  //WebMaker
  lightsSelect   : BOOL;
  socketsSelect  : BOOL;
  shuttersSelect : BOOL;
  AC_Select      : BOOL;
  navSelect      : usint;

  //RCU
  RCU_ethAdr   : TRemoteEthAdr;
  RCU_IP : TIPadr := [192, 168, 0, 23];
  RCU_Ch_localPort : UINT;
  Set_IP           : BOOL;
  GetAllStatus  : BOOL;
  SendIamServer : BOOL;

  //controlRoom
  controlRoom   : fbControlRoom ;
  lightsOutputDevs     : TlightsOutputDevs     := [(DevAddress := 1 , loopAddress := 1),(DevAddress := 1 , loopAddress := 2),
                                                   (DevAddress := 1 , loopAddress := 3),(DevAddress := 1 , loopAddress := 4),
                                                   (DevAddress := 1 , loopAddress := 5)];

  outletOutputDevs     : ToutletOutputDevs     := [(DevAddress := 1 , loopAddress := 6)];

  curtainsUpOutputDevs : TcurtainsUpOutputDevs := [(DevAddress := 1 , loopAddress := 8)];
  curtainsDwOutputDevs : TcurtainsDwOutputDevs := [(DevAddress := 1 , loopAddress := 9)];

  motionSensOutputDevs : TMotionSensOutputDevs := [(DevAddress := 1 , loopAddress := 1),(DevAddress := 1 , loopAddress := 2)];

  EnLights                            : TEnLights     ;
  EnLightsAN       {PUBLIC_API}       : TEnLightsAN   ;
  EnOutlets                           : TEnOutlets    ;
  EnOutletsAN      {PUBLIC_API}       : TEnOutletsAN  ;

  //
  enLights_RT  : Array[1..NumOfHMIsRoom1,1..NumOfLightRoom1] of R_TRIG;
  enLights_FT  : Array[1..NumOfHMIsRoom1,1..NumOfLightRoom1] of F_TRIG;

  enOutlets_RT : Array[1..NumOfHMIsRoom1,1..NumOfOutletRoom1] of R_TRIG;
  enOutlets_FT : Array[1..NumOfHMIsRoom1,1..NumOfOutletRoom1] of F_TRIG;

  // HMIs
  enCurtainsUP_RT : Array[1..NumOfHMIsRoom1,1..NumOfCurtainRoom1] of R_TRIG;
  enCurtainsUP_FT : Array[1..NumOfHMIsRoom1,1..NumOfCurtainRoom1] of F_TRIG;

  enCurtainsDW_RT : Array[1..NumOfHMIsRoom1,1..NumOfCurtainRoom1] of R_TRIG;
  enCurtainsDW_FT : Array[1..NumOfHMIsRoom1,1..NumOfCurtainRoom1] of F_TRIG;

  // RCU Switches
  enCurtainsUP_SW_RT : Array[1..NumOfCurtainRoom1] of R_TRIG;
  enCurtainsUP_SW_FT : Array[1..NumOfCurtainRoom1] of F_TRIG;

  enCurtainsDW_SW_RT : Array[1..NumOfCurtainRoom1] of R_TRIG;
  enCurtainsDW_SW_FT : Array[1..NumOfCurtainRoom1] of F_TRIG;

  // GUI
  enCurtainsUP_GUI : Array[1..NumOfCurtainRoom1] of BOOL;
  enCurtainsDW_GUI : Array[1..NumOfCurtainRoom1] of BOOL;

  CurtStatus_Index : USINT;
  CurtEn_Index     : USINT;

  //
  i , j : USINT;
  afterRestart_TP : TP;
  afterRestart_TP_FT : F_TRIG;

  //
  motionSensStatus                : TMotionSensStatus;
  CurtainsUpStatus   {PUBLIC_API} : TCurtainsUpStatus;
  CurtainsDwStatus   {PUBLIC_API} : TCurtainsDwStatus;

  // FCU VARS
  FCU          : Array[1..NumOfFCUsRoom1] of fbControlFCU;
  enableFCU    : Array[1..NumOfFCUsRoom1] of BOOL;
  settingsFCU  : Array[1..NumOfFCUsRoom1] of TFCU_Settings;

  //modeFCU      : Array[1..NumOfFCUsRoom1] of TFCU_Mode;
  //fanSpeedFCU  : Array[1..NumOfFCUsRoom1] of TFCU_FanSpeed;

  enFCUs_FT    : Array[1..NumOfHMIsRoom1,1..NumOfFCUsRoom1] of F_TRIG;
  enFCUs_RT    : Array[1..NumOfHMIsRoom1,1..NumOfFCUsRoom1] of R_TRIG;

  enFanHigh_RT : Array[1..NumOfHMIsRoom1,1..NumOfFCUsRoom1] of R_TRIG;
  enFanMed_RT  : Array[1..NumOfHMIsRoom1,1..NumOfFCUsRoom1] of R_TRIG;
  enFanLow_RT  : Array[1..NumOfHMIsRoom1,1..NumOfFCUsRoom1] of R_TRIG;
  enFanAuto_RT : Array[1..NumOfHMIsRoom1,1..NumOfFCUsRoom1] of R_TRIG;

  enFCUCool_RT    : Array[1..NumOfHMIsRoom1,1..NumOfFCUsRoom1] of R_TRIG;
  enFCUFanOnly_RT : Array[1..NumOfHMIsRoom1,1..NumOfFCUsRoom1] of R_TRIG;

  enSetTempIncr_RT : Array[1..NumOfHMIsRoom1,1..NumOfFCUsRoom1] of R_TRIG;
  enSetTempIncr_FT : Array[1..NumOfHMIsRoom1,1..NumOfFCUsRoom1] of F_TRIG;

  enSetTempDecr_RT : Array[1..NumOfHMIsRoom1,1..NumOfFCUsRoom1] of R_TRIG;
  enSetTempDecr_FT : Array[1..NumOfHMIsRoom1,1..NumOfFCUsRoom1] of F_TRIG;

  // config
  HMI_Index        : USINT;
  RCU_Index        : USINT;
  HMI_Addresses    : Array[1..NumOfHMIsRoom1] of USINT := [16, 17];

  END_VAR

   if navSelect = 0 then
     lightsSelect   := 1;
     socketsSelect  := 0;
     shuttersSelect := 0;
     AC_Select      := 0;
  elsif navSelect = 1 then
     lightsSelect   := 0;
     socketsSelect  := 1;
     shuttersSelect := 0;
     AC_Select      := 0;
  elsif navSelect = 2 then
     lightsSelect   := 0;
     socketsSelect  := 0;
     shuttersSelect := 1;
     AC_Select      := 0;
  elsif navSelect = 3 then
     lightsSelect   := 0;
     socketsSelect  := 0;
     shuttersSelect := 0;
     AC_Select      := 1;
  end_if;

  HMI_Index := 5;
  RCU_Index := 3;
  CurtStatus_Index := 6;
  CurtEn_Index  := 6;

  if GetRemoteIPaddress(chanCode := Eth1_uni2, ethAdr := RCU_ethAdr) then
     RCUs_IPs[RCU_Index] := RCU_ethAdr.remoteIP;
  end_if;

  HMIs_Info[HMI_Index].SNo := HMI_Addresses[1];
  HMIs_Info[HMI_Index].readStAdd  := 911;
  HMIs_Info[HMI_Index].writeStAdd := 971;
  HMIs_Info[HMI_Index].readNoPoint  := SIZEOF(HMIs_DataRead[HMI_Index]) / 2;
  HMIs_Info[HMI_Index].writeNoPoint := SIZEOF(HMIs_DataWrite[HMI_Index]) / 2;

  for i := 1 to NumOfHMIsRoom1-1 do
    HMIs_Info[HMI_Index+i] := HMIs_Info[HMI_Index];
    HMIs_Info[HMI_Index+i].SNo := HMI_Addresses[i+1];
  end_for;

  afterRestart_TP(IN := IS_COLD_RESTART_PLC or IS_HOT_RESTART_PLC, PT := T#2s );
  afterRestart_TP_FT(CLK := afterRestart_TP.Q);

  if afterRestart_TP_FT.Q then
     SendIamServer := 1;
  end_if;

  controlRoom(RCU_ChCode := ETH1_uni2 , RCU_PingDone := RCUs_PingDone[RCU_Index],
              numOfLights := NumOfLightRoom1 , numOfOutlets := NumOfOutletRoom1 , numOfCurtains := NumOfCurtainRoom1, numOfMotionSens := NumOfMotionSensRoom1,
              lightsOutputDevs := lightsOutputDevs , outletOutputDevs := outletOutputDevs ,
              curtainsUpOutputDevs := curtainsUpOutputDevs , curtainsDwOutputDevs := curtainsDwOutputDevs,
              RCU_CH_IN := void(ETH1_uni2_IN) , LightsStatus := lightsStatusRoom1 ,OutletsStatus := outletsStatusRoom1, MotionSenStatus := motionSensStatus,
              EnLights := EnLights , EnLightsAN := EnLightsAN , EnOutlets := EnOutlets ,EnOutletsAN :=EnOutletsAN ,
              SendIamServer := SendIamServer , GetAllStatus := GetAllStatus);

   FCU[1](enable := enableFCU[1], mode := settingsFCU[1].FCU_Mode, fanSpeed := settingsFCU[1].FCU_FanSpeed, setTemp := setTempFCU_Room1[1], temp := FCU_Temp_Room1, valve := FCU_valve_Room1, fanLow := FCU_fanLow_Room1,
                 fanMed := FCU_fanMed_Room1, fanHigh := FCU_fanHigh_Room1);

   for i := 1 to NumOfLightRoom1 do
       HMIs_DataWrite[HMI_Index].lightsStatus[i] := BOOL_TO_WORD(lightsStatusRoom1[i]);
   end_for;

   for i := 1 to NumOfOutletRoom1 do
       HMIs_DataWrite[HMI_Index].outletsStatus[i] := BOOL_TO_WORD(outletsStatusRoom1[i]);
   end_for;

   for i := 1 to NumOfMotionSensRoom1 do
       HMIs_DataWrite[HMI_Index].motionSensStatus[i] := BOOL_TO_WORD(motionSensStatus[i]);
   end_for;

   for i := 1 to NumOfFCUsRoom1 do
      HMIs_DataWrite[HMI_Index].FCUs_Status[i] := FCU[i].FCU_Status;
   end_for;

   if NumOfCurtainRoom1 > 0 then
      for i := 1 to NumOfCurtainRoom1 do
          HMIs_DataWrite[HMI_Index].shuttersStatus[i].UP.0 := curtainsStatus[CurtStatus_Index - 1 + i].outUP;
          HMIs_DataWrite[HMI_Index].shuttersStatus[i].Dw.0 := curtainsStatus[CurtStatus_Index - 1 + i].outDW;
          HMIs_DataWrite[HMI_Index].shuttersStatus[i].pos  := USINT_TO_WORD(curtainsStatus[CurtStatus_Index - 1 + i].normPos);
      end_for;
   end_if;

   for i := 1 to NumOfHMIsRoom1-1 do
     HMIs_DataWrite[HMI_Index+i] := HMIs_DataWrite[HMI_Index];
   end_for;

   for j := 1 to NumOfHMIsRoom1 do
     for i := 1 to NumOfLightRoom1 do

         enLights_RT[j,i](CLK := HMIs_DataRead[HMI_Index + j - 1].enLights[i]);

         enLights_FT[j,i](CLK := HMIs_DataRead[HMI_Index + j - 1].enLights[i]);

         if enLights_RT[j,i].Q or enLights_FT[j,i].Q then
            EnLights[i] := 1;
         end_if;
     end_for;
   end_for;

   for j := 1 to NumOfHMIsRoom1 do
     for i := 1 to NumOfOutletRoom1 do

         enOutlets_RT[j,i](CLK := HMIs_DataRead[HMI_Index + j - 1].enOutlets[i]);

         enOutlets_FT[j,i](CLK := HMIs_DataRead[HMI_Index + j - 1].enOutlets[i]);

         if enOutlets_RT[j,i].Q or enOutlets_FT[j,i].Q then
            EnOutlets[i] := 1;
         end_if;
     end_for;
   end_for;

   for j := 1 to NumOfHMIsRoom1 do
     for i := 1 to NumOfCurtainRoom1 do

         enCurtainsUP_RT[j,i](CLK := HMIs_DataRead[HMI_Index + j - 1].enShutters[i].UP.0);

         enCurtainsUP_FT[j,i](CLK := HMIs_DataRead[HMI_Index + j - 1].enShutters[i].UP.0);

         enCurtainsDW_RT[j,i](CLK := HMIs_DataRead[HMI_Index + j - 1].enShutters[i].Dw.0);

         enCurtainsDW_FT[j,i](CLK := HMIs_DataRead[HMI_Index + j - 1].enShutters[i].Dw.0);

         //
         enCurtainsUP_SW_RT[i](CLK := controlRoom.SwitchUPStatus[i]);
         enCurtainsUP_SW_FT[i](CLK := controlRoom.SwitchUPStatus[i]);

         enCurtainsDW_SW_RT[i](CLK := controlRoom.SwitchDWStatus[i]);
         enCurtainsDW_SW_FT[i](CLK := controlRoom.SwitchDWStatus[i]);

         if  enCurtainsUP_RT[j,i].Q  or enCurtainsUP_FT[j,i].Q or enCurtainsUP_SW_RT[i].Q or enCurtainsUP_SW_FT[i].Q then
             enCurtainsUP_GUI[i] := 1;
         end_if;

         if  enCurtainsDW_RT[j,i].Q  or enCurtainsDW_FT[j,i].Q or enCurtainsDW_SW_RT[i].Q or enCurtainsDW_SW_FT[i].Q then
             enCurtainsDW_GUI[i] := 1;
         end_if;

         // if up button is pressed and the curtain is not moving up

         if enCurtainsUP_GUI[i] and not curtainsStatus[CurtStatus_Index - 1 + i].outUP then
             PLC1_EnCurtains[CurtEn_Index - 1 + i].UP   := 1;
             PLC1_EnCurtains[CurtEn_Index - 1 + i].DW   := 0;
             PLC1_EnCurtains[CurtEn_Index - 1 + i].STOP := 0;

             enCurtainsUP_GUI[i] := 0;
         end_if;

         // if up button is pressed and the curtain is moving up

         if enCurtainsUP_GUI[i] and curtainsStatus[CurtStatus_Index - 1 + i].outUP then
             PLC1_EnCurtains[CurtEn_Index - 1 + i].UP   := 0;
             PLC1_EnCurtains[CurtEn_Index - 1 + i].DW   := 0;
             PLC1_EnCurtains[CurtEn_Index - 1 + i].STOP := 1;

             enCurtainsUP_GUI[i] := 0;
         end_if;

          // if down button is pressed and the curtain is not moving down

         if enCurtainsDW_GUI[i] and not curtainsStatus[CurtStatus_Index - 1 + i].outDW then
             PLC1_EnCurtains[CurtEn_Index - 1 + i].UP   := 0;
             PLC1_EnCurtains[CurtEn_Index - 1 + i].DW   := 1;
             PLC1_EnCurtains[CurtEn_Index - 1 + i].STOP := 0;

             enCurtainsDW_GUI[i] := 0;
         end_if;

         // if down button is pressed and the curtain is moving down

         if enCurtainsDW_GUI[i] and curtainsStatus[CurtStatus_Index - 1 + i].outDW then
             PLC1_EnCurtains[CurtEn_Index - 1 + i].UP   := 0;
             PLC1_EnCurtains[CurtEn_Index - 1 + i].DW   := 0;
             PLC1_EnCurtains[CurtEn_Index - 1 + i].STOP := 1;

             enCurtainsDW_GUI[i] := 0;
         end_if;

     end_for;
   end_for;

   for j := 1 to NumOfHMIsRoom1 do
      for i := 1 to NumOfFCUsRoom1 do
          enFCUs_FT[j,i](CLK := HMIs_DataRead[HMI_Index + j - 1].enFCUs[i].onOff);
          enFCUs_RT[j,i](CLK := HMIs_DataRead[HMI_Index + j - 1].enFCUs[i].onOff);

          if enFCUs_FT[j,i].Q then
             enableFCU[i] := 0;
          end_if;
          if enFCUs_RT[j,i].Q then
             enableFCU[i] := 1;
          end_if;

          enFanAuto_RT[j,i](CLK := (HMIs_DataRead[HMI_Index + j - 1].enFCUs[i].fanSpeed = 8));
          enFanLow_RT[j,i](CLK := HMIs_DataRead[HMI_Index + j - 1].enFCUs[i].fanSpeed.0);
          enFanMed_RT[j,i](CLK := HMIs_DataRead[HMI_Index + j - 1].enFCUs[i].fanSpeed.1);
          enFanHigh_RT[j,i](CLK := HMIs_DataRead[HMI_Index + j - 1].enFCUs[i].fanSpeed.2);

          if enFanAuto_RT[j,i].Q then
             settingsFCU[i].FCU_FanSpeed := auto;
          end_if;
          if enFanLow_RT[j,i].Q then
             settingsFCU[i].FCU_FanSpeed := low;
          end_if;
          if enFanMed_RT[j,i].Q then
             settingsFCU[i].FCU_FanSpeed := med;
          end_if;
          if enFanHigh_RT[j,i].Q then
             settingsFCU[i].FCU_FanSpeed := high;
          end_if;

          enFCUCool_RT[j,i](CLK := (HMIs_DataRead[HMI_Index + j - 1].enFCUs[i].mode = 0));
          enFCUFanOnly_RT[j,i](CLK := HMIs_DataRead[HMI_Index + j - 1].enFCUs[i].mode.0);

          if enFCUCool_RT[j,i].Q then
             settingsFCU[i].FCU_Mode := cooling;
          end_if;
          if enFCUFanOnly_RT[j,i].Q then
             settingsFCU[i].FCU_Mode := fanOnly;
          end_if;

          enSetTempIncr_RT[j,i](CLK := HMIs_DataRead[HMI_Index + j - 1].enFCUs[i].SetTempCtrl.0);
          enSetTempIncr_FT[j,i](CLK := HMIs_DataRead[HMI_Index + j - 1].enFCUs[i].SetTempCtrl.0);

          if enSetTempIncr_RT[j,i].Q or enSetTempIncr_FT[j,i].Q then
             setTempFCU_Room1[j] := setTempFCU_Room1[j] + 0.5;
          end_if;

          enSetTempDecr_RT[j,i](CLK := HMIs_DataRead[HMI_Index + j - 1].enFCUs[i].SetTempCtrl.1);
          enSetTempDecr_FT[j,i](CLK := HMIs_DataRead[HMI_Index + j - 1].enFCUs[i].SetTempCtrl.1);

          if enSetTempDecr_RT[j,i].Q or enSetTempDecr_FT[j,i].Q then
             setTempFCU_Room1[j] := setTempFCU_Room1[j] - 0.5;
          end_if;

      end_for;
   end_for;

END_PROGRAM

(* ---- PrgRoom2.ST ---- *)
VAR_GLOBAL CONSTANT
   NumOfLightRoom2      : USINT := 5;
   NumOfOutletRoom2     : USINT := 1;
   NumOfCurtainRoom2    : USINT := 1;
   NumOfMotionSensRoom2 : USINT := 2;
   NumOfFCUsRoom2       : USINT := 1;
   NumOfHMIsRoom2       : USINT := 2;
END_VAR

VAR_GLOBAL RETAIN
   lightsStatusRoom2  {PUBLIC_API} : TLightsStatus;
   outletsStatusRoom2 {PUBLIC_API} : TOutletsStatus;
   setTempFCU_Room2  : Array[1..NumOfFCUsRoom2] of REAL := [20];

END_VAR

PROGRAM PrgRoom2

  VAR
  //WebMaker
  lightsSelect   : BOOL;
  socketsSelect  : BOOL;
  shuttersSelect : BOOL;
  AC_Select      : BOOL;
  navSelect      : usint;

  //RCU
  RCU_ethAdr   : TRemoteEthAdr;
  RCU_IP : TIPadr := [192, 168, 0, 23];
  RCU_Ch_localPort : UINT;
  Set_IP           : BOOL;
  GetAllStatus  : BOOL;
  SendIamServer : BOOL;

  //controlRoom
  controlRoom   : fbControlRoom ;
  lightsOutputDevs     : TlightsOutputDevs     := [(DevAddress := 1 , loopAddress := 1),(DevAddress := 1 , loopAddress := 2),
                                                   (DevAddress := 1 , loopAddress := 3),(DevAddress := 1 , loopAddress := 4),
                                                   (DevAddress := 1 , loopAddress := 5)];

  outletOutputDevs     : ToutletOutputDevs     := [(DevAddress := 1 , loopAddress := 6)];

  curtainsUpOutputDevs : TcurtainsUpOutputDevs := [(DevAddress := 1 , loopAddress := 8)];
  curtainsDwOutputDevs : TcurtainsDwOutputDevs := [(DevAddress := 1 , loopAddress := 9)];

  motionSensOutputDevs : TMotionSensOutputDevs := [(DevAddress := 1 , loopAddress := 1),(DevAddress := 1 , loopAddress := 2)];

  EnLights                            : TEnLights     ;
  EnLightsAN       {PUBLIC_API}       : TEnLightsAN   ;
  EnOutlets                           : TEnOutlets    ;
  EnOutletsAN      {PUBLIC_API}       : TEnOutletsAN  ;
  EnCurtainsUp     {PUBLIC_API}       : TEnCurtainsUp ;
  EnCurtainsDw     {PUBLIC_API}       : TEnCurtainsDW ;

  //
  enLights_RT  : Array[1..NumOfHMIsRoom2,1..NumOfLightRoom2] of R_TRIG;
  enLights_FT  : Array[1..NumOfHMIsRoom2,1..NumOfLightRoom2] of F_TRIG;

  enOutlets_RT : Array[1..NumOfHMIsRoom2,1..NumOfOutletRoom2] of R_TRIG;
  enOutlets_FT : Array[1..NumOfHMIsRoom2,1..NumOfOutletRoom2] of F_TRIG;

  // HMIs
  enCurtainsUP_RT : Array[1..NumOfHMIsRoom2,1..NumOfCurtainRoom2] of R_TRIG;
  enCurtainsUP_FT : Array[1..NumOfHMIsRoom2,1..NumOfCurtainRoom2] of F_TRIG;

  enCurtainsDW_RT : Array[1..NumOfHMIsRoom2,1..NumOfCurtainRoom2] of R_TRIG;
  enCurtainsDW_FT : Array[1..NumOfHMIsRoom2,1..NumOfCurtainRoom2] of F_TRIG;

  // RCU Switches
  enCurtainsUP_SW_RT : Array[1..NumOfCurtainRoom2] of R_TRIG;
  enCurtainsUP_SW_FT : Array[1..NumOfCurtainRoom2] of F_TRIG;

  enCurtainsDW_SW_RT : Array[1..NumOfCurtainRoom2] of R_TRIG;
  enCurtainsDW_SW_FT : Array[1..NumOfCurtainRoom2] of F_TRIG;

  // GUI
  enCurtainsUP_GUI : Array[1..NumOfCurtainRoom2] of BOOL;
  enCurtainsDW_GUI : Array[1..NumOfCurtainRoom2] of BOOL;

  CurtStatus_Index : USINT;
  CurtEn_Index     : USINT;

  //
  i , j : USINT;
  afterRestart_TP : TP;
  afterRestart_TP_FT : F_TRIG;

  //
  motionSensStatus                : TMotionSensStatus;
  CurtainsUpStatus   {PUBLIC_API} : TCurtainsUpStatus;
  CurtainsDwStatus   {PUBLIC_API} : TCurtainsDwStatus;

  // FCU VARS
  FCU          : Array[1..NumOfFCUsRoom2] of fbControlFCU;
  enableFCU    : Array[1..NumOfFCUsRoom2] of BOOL;
  settingsFCU  : Array[1..NumOfFCUsRoom2] of TFCU_Settings;

  //modeFCU      : Array[1..NumOfFCUsRoom2] of TFCU_Mode;
  //fanSpeedFCU  : Array[1..NumOfFCUsRoom2] of TFCU_FanSpeed;

  enFCUs_FT    : Array[1..NumOfHMIsRoom2,1..NumOfFCUsRoom2] of F_TRIG;
  enFCUs_RT    : Array[1..NumOfHMIsRoom2,1..NumOfFCUsRoom2] of R_TRIG;

  enFanHigh_RT : Array[1..NumOfHMIsRoom2,1..NumOfFCUsRoom2] of R_TRIG;
  enFanMed_RT  : Array[1..NumOfHMIsRoom2,1..NumOfFCUsRoom2] of R_TRIG;
  enFanLow_RT  : Array[1..NumOfHMIsRoom2,1..NumOfFCUsRoom2] of R_TRIG;
  enFanAuto_RT : Array[1..NumOfHMIsRoom2,1..NumOfFCUsRoom2] of R_TRIG;

  enFCUCool_RT    : Array[1..NumOfHMIsRoom2,1..NumOfFCUsRoom2] of R_TRIG;
  enFCUFanOnly_RT : Array[1..NumOfHMIsRoom2,1..NumOfFCUsRoom2] of R_TRIG;

  enSetTempIncr_RT : Array[1..NumOfHMIsRoom2,1..NumOfFCUsRoom2] of R_TRIG;
  enSetTempIncr_FT : Array[1..NumOfHMIsRoom2,1..NumOfFCUsRoom2] of F_TRIG;

  enSetTempDecr_RT : Array[1..NumOfHMIsRoom2,1..NumOfFCUsRoom2] of R_TRIG;
  enSetTempDecr_FT : Array[1..NumOfHMIsRoom2,1..NumOfFCUsRoom2] of F_TRIG;

  //HMIs[1..num
  HMI_Index : USINT;
  RCU_Index : USINT;
  HMI_Addresses : Array[1..NumOfHMIsRoom2] of USINT := [18, 19];

  END_VAR

   if navSelect = 0 then
     lightsSelect   := 1;
     socketsSelect  := 0;
     shuttersSelect := 0;
     AC_Select      := 0;
  elsif navSelect = 1 then
     lightsSelect   := 0;
     socketsSelect  := 1;
     shuttersSelect := 0;
     AC_Select      := 0;
  elsif navSelect = 2 then
     lightsSelect   := 0;
     socketsSelect  := 0;
     shuttersSelect := 1;
     AC_Select      := 0;
  elsif navSelect = 3 then
     lightsSelect   := 0;
     socketsSelect  := 0;
     shuttersSelect := 0;
     AC_Select      := 1;
  end_if;

  HMI_Index := 7;
  RCU_Index := 4;
  CurtStatus_Index := 7;
  CurtEn_Index  := 7;

  if GetRemoteIPaddress(chanCode := Eth1_uni3, ethAdr := RCU_ethAdr) then
     RCUs_IPs[RCU_Index] := RCU_ethAdr.remoteIP;
  end_if;

  HMIs_Info[HMI_Index].SNo := HMI_Addresses[1];
  HMIs_Info[HMI_Index].readStAdd  := 1041;
  HMIs_Info[HMI_Index].writeStAdd := 1101;
  HMIs_Info[HMI_Index].readNoPoint  := SIZEOF(HMIs_DataRead[HMI_Index]) / 2;
  HMIs_Info[HMI_Index].writeNoPoint := SIZEOF(HMIs_DataWrite[HMI_Index]) / 2;

  for i := 1 to NumOfHMIsRoom2-1 do
    HMIs_Info[HMI_Index+i] := HMIs_Info[HMI_Index];
    HMIs_Info[HMI_Index+i].SNo := HMI_Addresses[i+1];
  end_for;

  afterRestart_TP(IN := IS_COLD_RESTART_PLC or IS_HOT_RESTART_PLC, PT := T#2s );
  afterRestart_TP_FT(CLK := afterRestart_TP.Q);

  if afterRestart_TP_FT.Q then
     SendIamServer := 1;
  end_if;

  controlRoom(RCU_ChCode := ETH1_uni3 , RCU_PingDone := RCUs_PingDone[RCU_Index],
              numOfLights := NumOfLightRoom2 , numOfOutlets := NumOfOutletRoom2 , numOfCurtains := NumOfCurtainRoom2, numOfMotionSens := NumOfMotionSensRoom2,
              lightsOutputDevs := lightsOutputDevs , outletOutputDevs := outletOutputDevs ,
              curtainsUpOutputDevs := curtainsUpOutputDevs , curtainsDwOutputDevs := curtainsDwOutputDevs,
              RCU_CH_IN := void(ETH1_uni3_IN) , LightsStatus := lightsStatusRoom2 ,OutletsStatus := outletsStatusRoom2, MotionSenStatus := motionSensStatus,
              EnLights := EnLights , EnLightsAN := EnLightsAN , EnOutlets := EnOutlets ,EnOutletsAN :=EnOutletsAN ,
              SendIamServer := SendIamServer , GetAllStatus := GetAllStatus);

              //stLightsRoom2AN := lightsStatusRoom2[1];

   FCU[1](enable := enableFCU[1], mode := settingsFCU[1].FCU_Mode, fanSpeed := settingsFCU[1].FCU_FanSpeed, setTemp := setTempFCU_Room2[1], temp := FCU_Temp_Room2, valve := FCU_valve_Room2, fanLow := FCU_fanLow_Room2,
                 fanMed := FCU_fanMed_Room2, fanHigh := FCU_fanHigh_Room2);

   for i := 1 to NumOfLightRoom2 do
       HMIs_DataWrite[HMI_Index].lightsStatus[i] := BOOL_TO_WORD(lightsStatusRoom2[i]);
   end_for;

   for i := 1 to NumOfOutletRoom2 do
       HMIs_DataWrite[HMI_Index].outletsStatus[i] := BOOL_TO_WORD(outletsStatusRoom2[i]);
   end_for;

   for i := 1 to NumOfMotionSensRoom2 do
       HMIs_DataWrite[HMI_Index].motionSensStatus[i] := BOOL_TO_WORD(motionSensStatus[i]);
   end_for;

   for i := 1 to NumOfFCUsRoom2 do
      HMIs_DataWrite[HMI_Index].FCUs_Status[i] := FCU[i].FCU_Status;
   end_for;

    if NumOfCurtainRoom2 > 0 then
      for i := 1 to NumOfCurtainRoom2 do
          HMIs_DataWrite[HMI_Index].shuttersStatus[i].UP.0 := curtainsStatus[CurtStatus_Index - 1 + i].outUP;
          HMIs_DataWrite[HMI_Index].shuttersStatus[i].Dw.0 := curtainsStatus[CurtStatus_Index - 1 + i].outDW;
          HMIs_DataWrite[HMI_Index].shuttersStatus[i].pos  := USINT_TO_WORD(curtainsStatus[CurtStatus_Index - 1 + i].pos);
      end_for;
   end_if;

   for i := 1 to NumOfHMIsRoom2-1 do
     HMIs_DataWrite[HMI_Index+i] := HMIs_DataWrite[HMI_Index];
   end_for;

   for j := 1 to NumOfHMIsRoom2 do
     for i := 1 to NumOfLightRoom2 do

         enLights_RT[j,i](CLK := HMIs_DataRead[HMI_Index + j - 1].enLights[i]);

         enLights_FT[j,i](CLK := HMIs_DataRead[HMI_Index + j - 1].enLights[i]);

         if enLights_RT[j,i].Q or enLights_FT[j,i].Q then
            EnLights[i] := 1;
         end_if;
     end_for;
   end_for;

   for j := 1 to NumOfHMIsRoom2 do
     for i := 1 to NumOfOutletRoom2 do

         enOutlets_RT[j,i](CLK := HMIs_DataRead[HMI_Index + j - 1].enOutlets[i]);

         enOutlets_FT[j,i](CLK := HMIs_DataRead[HMI_Index + j - 1].enOutlets[i]);

         if enOutlets_RT[j,i].Q or enOutlets_FT[j,i].Q then
            EnOutlets[i] := 1;
         end_if;
     end_for;
   end_for;

   for j := 1 to NumOfHMIsRoom2 do
     for i := 1 to NumOfCurtainRoom2 do

         enCurtainsUP_RT[j,i](CLK := HMIs_DataRead[HMI_Index + j - 1].enShutters[i].UP.0);

         enCurtainsUP_FT[j,i](CLK := HMIs_DataRead[HMI_Index + j - 1].enShutters[i].UP.0);

         enCurtainsDW_RT[j,i](CLK := HMIs_DataRead[HMI_Index + j - 1].enShutters[i].Dw.0);

         enCurtainsDW_FT[j,i](CLK := HMIs_DataRead[HMI_Index + j - 1].enShutters[i].Dw.0);

         //
         enCurtainsUP_SW_RT[i](CLK := controlRoom.SwitchUPStatus[i]);
         enCurtainsUP_SW_FT[i](CLK := controlRoom.SwitchUPStatus[i]);

         enCurtainsDW_SW_RT[i](CLK := controlRoom.SwitchDWStatus[i]);
         enCurtainsDW_SW_FT[i](CLK := controlRoom.SwitchDWStatus[i]);

         if  enCurtainsUP_RT[j,i].Q  or enCurtainsUP_FT[j,i].Q then
             enCurtainsUP_GUI[i] := 1;
         end_if;

         if  enCurtainsDW_RT[j,i].Q  or enCurtainsDW_FT[j,i].Q then
             enCurtainsDW_GUI[i] := 1;
         end_if;

         // if up button is pressed and the curtain is not moving up

         if (enCurtainsUP_GUI[i] or enCurtainsUP_SW_RT[i].Q) and not curtainsStatus[CurtStatus_Index - 1 + i].outUP then
             PLC1_EnCurtains[CurtEn_Index - 1 + i].UP   := 1;
             PLC1_EnCurtains[CurtEn_Index - 1 + i].DW   := 0;
             PLC1_EnCurtains[CurtEn_Index - 1 + i].STOP := 0;

             enCurtainsUP_GUI[i] := 0;
         end_if;

         // if up button is pressed and the curtain is moving up

         if (enCurtainsUP_GUI[i] or enCurtainsUP_SW_FT[i].Q) and curtainsStatus[CurtStatus_Index - 1 + i].outUP then
             PLC1_EnCurtains[CurtEn_Index - 1 + i].UP   := 0;
             PLC1_EnCurtains[CurtEn_Index - 1 + i].DW   := 0;
             PLC1_EnCurtains[CurtEn_Index - 1 + i].STOP := 1;

             enCurtainsUP_GUI[i] := 0;
         end_if;

          // if down button is pressed and the curtain is not moving down

         if (enCurtainsDW_GUI[i] or enCurtainsDW_SW_RT[i].Q) and not curtainsStatus[CurtStatus_Index - 1 + i].outDW then
             PLC1_EnCurtains[CurtEn_Index - 1 + i].UP   := 0;
             PLC1_EnCurtains[CurtEn_Index - 1 + i].DW   := 1;
             PLC1_EnCurtains[CurtEn_Index - 1 + i].STOP := 0;

             enCurtainsDW_GUI[i] := 0;
         end_if;

         // if down button is pressed and the curtain is moving down

         if (enCurtainsDW_GUI[i] or enCurtainsDW_SW_FT[i].Q) and curtainsStatus[CurtStatus_Index - 1 + i].outDW then
             PLC1_EnCurtains[CurtEn_Index - 1 + i].UP   := 0;
             PLC1_EnCurtains[CurtEn_Index - 1 + i].DW   := 0;
             PLC1_EnCurtains[CurtEn_Index - 1 + i].STOP := 1;

             enCurtainsDW_GUI[i] := 0;
         end_if;

     end_for;
   end_for;

   for j := 1 to NumOfHMIsRoom2 do
      for i := 1 to NumOfFCUsRoom2 do
          enFCUs_FT[j,i](CLK := HMIs_DataRead[HMI_Index + j - 1].enFCUs[i].onOff);
          enFCUs_RT[j,i](CLK := HMIs_DataRead[HMI_Index + j - 1].enFCUs[i].onOff);

          if enFCUs_FT[j,i].Q then
             enableFCU[i] := 0;
          end_if;
          if enFCUs_RT[j,i].Q then
             enableFCU[i] := 1;
          end_if;

          enFanAuto_RT[j,i](CLK := (HMIs_DataRead[HMI_Index + j - 1].enFCUs[i].fanSpeed = 8));
          enFanLow_RT[j,i](CLK := HMIs_DataRead[HMI_Index + j - 1].enFCUs[i].fanSpeed.0);
          enFanMed_RT[j,i](CLK := HMIs_DataRead[HMI_Index + j - 1].enFCUs[i].fanSpeed.1);
          enFanHigh_RT[j,i](CLK := HMIs_DataRead[HMI_Index + j - 1].enFCUs[i].fanSpeed.2);

          if enFanAuto_RT[j,i].Q then
             settingsFCU[i].FCU_FanSpeed := auto;
          end_if;
          if enFanLow_RT[j,i].Q then
             settingsFCU[i].FCU_FanSpeed := low;
          end_if;
          if enFanMed_RT[j,i].Q then
             settingsFCU[i].FCU_FanSpeed := med;
          end_if;
          if enFanHigh_RT[j,i].Q then
             settingsFCU[i].FCU_FanSpeed := high;
          end_if;

          enFCUCool_RT[j,i](CLK := (HMIs_DataRead[HMI_Index + j - 1].enFCUs[i].mode = 0));
          enFCUFanOnly_RT[j,i](CLK := HMIs_DataRead[HMI_Index + j - 1].enFCUs[i].mode.0);

          if enFCUCool_RT[j,i].Q then
             settingsFCU[i].FCU_Mode := cooling;
          end_if;
          if enFCUFanOnly_RT[j,i].Q then
             settingsFCU[i].FCU_Mode := fanOnly;
          end_if;

          enSetTempIncr_RT[j,i](CLK := HMIs_DataRead[HMI_Index + j - 1].enFCUs[i].SetTempCtrl.0);
          enSetTempIncr_FT[j,i](CLK := HMIs_DataRead[HMI_Index + j - 1].enFCUs[i].SetTempCtrl.0);

          if enSetTempIncr_RT[j,i].Q or enSetTempIncr_FT[j,i].Q then
             setTempFCU_Room2[j] := setTempFCU_Room2[j] + 0.5;
          end_if;

          enSetTempDecr_RT[j,i](CLK := HMIs_DataRead[HMI_Index + j - 1].enFCUs[i].SetTempCtrl.1);
          enSetTempDecr_FT[j,i](CLK := HMIs_DataRead[HMI_Index + j - 1].enFCUs[i].SetTempCtrl.1);

          if enSetTempDecr_RT[j,i].Q or enSetTempDecr_FT[j,i].Q then
             setTempFCU_Room2[j] := setTempFCU_Room2[j] - 0.5;
          end_if;

      end_for;
   end_for;

END_PROGRAM
